LIN {X 0,Y 266.762,Z 400.732,A -85,B 0,C 180,E1 -19209.692,E2 -19209.692} C_VEL
LIN {X 0,Y 260.69,Z 388.855,A -85,B 0,C 180,E1 -19211.354,E2 -19211.354} C_VEL
LIN {X 0,Y 253.783,Z 376.661,A -85,B 0,C 180,E1 -19213.353,E2 -19213.353} C_VEL
LIN {X 0,Y 250.06,Z 370.765,A -85,B 0,C 180,E1 -19214.482,E2 -19214.482} C_VEL
LIN {X 0,Y 247.221,Z 366.216,A -85,B 0,C 180,E1 -19215.384,E2 -19215.384} C_VEL
LIN {X 0,Y 244.284,Z 361.418,A -85,B 0,C 180,E1 -19216.424,E2 -19216.424} C_VEL
LIN {X 0,Y 241.94,Z 353.971,A -85,B 0,C 180,E1 -19220.655,E2 -19220.655} C_VEL
LIN {X 0,Y 241.982,Z 353.963,A -85,B 0,C 180,E1 -19224.489,E2 -19224.489} C_VEL
LIN {X 0,Y 241.941,Z 353.945,A -85,B 0,C 180,E1 -19228.476,E2 -19228.476} C_VEL
LIN {X 0,Y 241.954,Z 353.955,A -85,B 0,C 180,E1 -19232.306,E2 -19232.306} C_VEL
LIN {X 0,Y 242.018,Z 353.954,A -85,B 0,C 180,E1 -19236.012,E2 -19236.012} C_VEL
LIN {X 0,Y 242.013,Z 353.953,A -85,B 0,C 180,E1 -19239.606,E2 -19239.606} C_VEL
LIN {X 0,Y 242.109,Z 353.941,A -85,B 0,C 180,E1 -19243.316,E2 -19243.316} C_VEL
LIN {X 0,Y 242.128,Z 353.949,A -85,B 0,C 180,E1 -19246.573,E2 -19246.573} C_VEL
LIN {X 0,Y 242.36,Z 353.915,A -85,B 0,C 180,E1 -19251.664,E2 -19251.664} C_VEL
LIN {X 0,Y 242.387,Z 353.904,A -85,B 0,C 180,E1 -19253.34,E2 -19253.34} C_VEL
LIN {X 0,Y 242.612,Z 353.876,A -85,B 0,C 180,E1 -19258.341,E2 -19258.341} C_VEL
LIN {X 0,Y 242.612,Z 353.88,A -85,B 0,C 180,E1 -19261.661,E2 -19261.661} C_VEL
LIN {X 0,Y 242.398,Z 353.906,A -85,B 0,C 180,E1 -19266.66,E2 -19266.66} C_VEL
LIN {X 0,Y 242.256,Z 353.934,A -85,B 0,C 180,E1 -19270.025,E2 -19270.025} C_VEL
LIN {X 0,Y 242.116,Z 353.947,A -85,B 0,C 180,E1 -19275.145,E2 -19275.145} C_VEL
LIN {X 0,Y 242.026,Z 353.963,A -85,B 0,C 180,E1 -19278.629,E2 -19278.629} C_VEL
LIN {X 0,Y 241.997,Z 353.965,A -85,B 0,C 180,E1 -19282.182,E2 -19282.182} C_VEL
LIN {X 0,Y 242.063,Z 353.956,A -85,B 0,C 180,E1 -19285.839,E2 -19285.839} C_VEL
LIN {X 0,Y 242.026,Z 353.963,A -85,B 0,C 180,E1 -19289.582,E2 -19289.582} C_VEL
LIN {X 0,Y 241.978,Z 353.965,A -85,B 0,C 180,E1 -19293.494,E2 -19293.494} C_VEL
LIN {X 0,Y 242.004,Z 354.056,A -85,B 0,C 180,E1 -19297.122,E2 -19297.122} C_VEL
LIN {X 0,Y 242.918,Z 356.668,A -85,B 0,C 180,E1 -19297.493,E2 -19297.493} C_VEL
LIN {X 0,Y 245.113,Z 359.008,A -85,B 0,C 180,E1 -19298.192,E2 -19298.192} C_VEL
LIN {X 0,Y 247.682,Z 362.902,A -85,B 0,C 180,E1 -19299.03,E2 -19299.03} C_VEL
LIN {X 0,Y 249.024,Z 364.607,A -85,B 0,C 180,E1 -19299.442,E2 -19299.442} C_VEL
LIN {X 0,Y 255.386,Z 373.693,A -85,B 0,C 180,E1 -19301.336,E2 -19301.336} C_VEL
LIN {X 0,Y 262.149,Z 384.884,A -85,B 0,C 180,E1 -19303.241,E2 -19303.241} C_VEL
LIN {X 0,Y 270.133,Z 399.946,A -85,B 0,C 180,E1 -19305.361,E2 -19305.361} C_VEL
LIN {X 0,Y 275.739,Z 412.188,A -85,B 0,C 180,E1 -19306.793,E2 -19306.793} C_VEL
LIN {X 0,Y 271.981,Z 488.618,A -85,B 0,C 180,E1 -19308.739,E2 -19308.739} C_VEL
LIN {X 0,Y 270.539,Z 503.215,A -85,B 0,C 180,E1 -19309.389,E2 -19309.389} C_VEL
LIN {X 0,Y 268.489,Z 517.743,A -85,B 0,C 180,E1 -19310.355,E2 -19310.355} C_VEL
LIN {X 0,Y 266.247,Z 529.779,A -85,B 0,C 180,E1 -19311.42,E2 -19311.42} C_VEL
LIN {X 0,Y 263.578,Z 541.335,A -85,B 0,C 180,E1 -19312.705,E2 -19312.705} C_VEL
LIN {X 0,Y 260.501,Z 552.94,A -85,B 0,C 180,E1 -19314.328,E2 -19314.328} C_VEL
LIN {X 0,Y 257.523,Z 562.64,A -85,B 0,C 180,E1 -19315.983,E2 -19315.983} C_VEL
LIN {X 0,Y 254.098,Z 573.453,A -85,B 0,C 180,E1 -19318.298,E2 -19318.298} C_VEL
LIN {X 0,Y 251.147,Z 582.347,A -85,B 0,C 180,E1 -19320.679,E2 -19320.679} C_VEL
LIN {X 0,Y 248.431,Z 589.714,A -85,B 0,C 180,E1 -19323.088,E2 -19323.088} C_VEL
LIN {X 0,Y 246.113,Z 595.823,A -85,B 0,C 180,E1 -19325.54,E2 -19325.54} C_VEL
LIN {X 0,Y 244.196,Z 600.861,A -85,B 0,C 180,E1 -19328.029,E2 -19328.029} C_VEL
LIN {X 0,Y 242.228,Z 606.023,A -85,B 0,C 180,E1 -19331.389,E2 -19331.389} C_VEL
LIN {X 0,Y 240.942,Z 609.649,A -85,B 0,C 180,E1 -19334.781,E2 -19334.781} C_VEL
LIN {X 0,Y 240.025,Z 611.858,A -85,B 0,C 180,E1 -19338.173,E2 -19338.173} C_VEL
LIN {X 0,Y 239.773,Z 612.71,A -85,B 0,C 180,E1 -19341.573,E2 -19341.573} C_VEL
LIN {X 0,Y 239.848,Z 612.21,A -85,B 0,C 180,E1 -19345.056,E2 -19345.056} C_VEL
LIN {X 0,Y 239.95,Z 610.455,A -85,B 0,C 180,E1 -19348.322,E2 -19348.322} C_VEL
LIN {X 0,Y 240.27,Z 607.324,A -85,B 0,C 180,E1 -19351.676,E2 -19351.676} C_VEL
LIN {X 0,Y 241.059,Z 602.721,A -85,B 0,C 180,E1 -19355.018,E2 -19355.018} C_VEL
LIN {X 0,Y 242.464,Z 596.49,A -85,B 0,C 180,E1 -19358.333,E2 -19358.333} C_VEL
LIN {X 0,Y 244.301,Z 589.549,A -85,B 0,C 180,E1 -19361.197,E2 -19361.197} C_VEL
LIN {X 0,Y 246.354,Z 581.698,A -85,B 0,C 180,E1 -19363.802,E2 -19363.802} C_VEL
LIN {X 0,Y 248.233,Z 573.619,A -85,B 0,C 180,E1 -19366.024,E2 -19366.024} C_VEL
LIN {X 0,Y 250.756,Z 563.089,A -85,B 0,C 180,E1 -19368.379,E2 -19368.379} C_VEL
LIN {X 0,Y 253.22,Z 552.45,A -85,B 0,C 180,E1 -19370.299,E2 -19370.299} C_VEL
LIN {X 0,Y 255.525,Z 540.847,A -85,B 0,C 180,E1 -19372.008,E2 -19372.008} C_VEL
LIN {X 0,Y 257.784,Z 528.072,A -85,B 0,C 180,E1 -19373.498,E2 -19373.498} C_VEL
LIN {X 0,Y 259.576,Z 515.909,A -85,B 0,C 180,E1 -19374.599,E2 -19374.599} C_VEL
LIN {X 0,Y 261.232,Z 501.809,A -85,B 0,C 180,E1 -19375.549,E2 -19375.549} C_VEL
LIN {X 0,Y 262.272,Z 488.028,A -85,B 0,C 180,E1 -19376.186,E2 -19376.186} C_VEL
LIN {X 0,Y 265.58,Z 403.027,A -85,B 0,C 180,E1 -19378.445,E2 -19378.445} C_VEL
LIN {X 0,Y 263.893,Z 398.103,A -85,B 0,C 180,E1 -19378.83,E2 -19378.83} C_VEL
LIN {X 0,Y 257.563,Z 382.943,A -85,B 0,C 180,E1 -19380.226,E2 -19380.226} C_VEL
LIN {X 0,Y 251.704,Z 370.899,A -85,B 0,C 180,E1 -19381.533,E2 -19381.533} C_VEL
LIN {X 0,Y 243.648,Z 357.672,A -85,B 0,C 180,E1 -19383.35,E2 -19383.35} C_VEL
LIN {X 0,Y 242.306,Z 355.295,A -85,B 0,C 180,E1 -19383.675,E2 -19383.675} C_VEL
LIN {X 0,Y 242.016,Z 353.964,A -85,B 0,C 180,E1 -19383.796,E2 -19383.796} C_VEL
LIN {X 0,Y 242.003,Z 353.966,A -85,B 0,C 180,E1 -19387.578,E2 -19387.578} C_VEL
LIN {X 0,Y 241.938,Z 353.961,A -85,B 0,C 180,E1 -19391.921,E2 -19391.921} C_VEL
LIN {X 0,Y 241.926,Z 353.975,A -85,B 0,C 180,E1 -19396.572,E2 -19396.572} C_VEL
LIN {X 0,Y 241.954,Z 353.971,A -85,B 0,C 180,E1 -19400.279,E2 -19400.279} C_VEL
LIN {X 0,Y 241.984,Z 353.967,A -85,B 0,C 180,E1 -19404.488,E2 -19404.488} C_VEL
LIN {X 0,Y 241.969,Z 353.967,A -85,B 0,C 180,E1 -19408.478,E2 -19408.478} C_VEL
LIN {X 0,Y 241.986,Z 353.946,A -85,B 0,C 180,E1 -19412.309,E2 -19412.309} C_VEL
LIN {X 0,Y 242.032,Z 353.961,A -85,B 0,C 180,E1 -19416.013,E2 -19416.013} C_VEL
LIN {X 0,Y 241.987,Z 353.941,A -85,B 0,C 180,E1 -19419.603,E2 -19419.603} C_VEL
LIN {X 0,Y 242.108,Z 353.952,A -85,B 0,C 180,E1 -19423.317,E2 -19423.317} C_VEL
LIN {X 0,Y 242.157,Z 353.922,A -85,B 0,C 180,E1 -19428.278,E2 -19428.278} C_VEL
LIN {X 0,Y 242.379,Z 353.917,A -85,B 0,C 180,E1 -19431.663,E2 -19431.663} C_VEL
LIN {X 0,Y 242.4,Z 353.906,A -85,B 0,C 180,E1 -19433.34,E2 -19433.34} C_VEL
LIN {X 0,Y 242.61,Z 353.884,A -85,B 0,C 180,E1 -19438.339,E2 -19438.339} C_VEL
LIN {X 0,Y 242.6,Z 353.887,A -85,B 0,C 180,E1 -19439.548,E2 -19439.548} C_VEL
LIN {X 0,Y 241.968,Z 353.976,A -85,B 0,C 180,E1 -19440.929,E2 -19440.929} C_VEL
LIN {X 0,Y 239.092,Z 354.347,A -85,B 0,C 180,E1 -19443.179,E2 -19443.179} C_VEL
LIN {X 0,Y 236.583,Z 354.657,A -85,B 0,C 180,E1 -19445.011,E2 -19445.011} C_VEL
LIN {X 0,Y 235.452,Z 354.786,A -85,B 0,C 180,E1 -19446.436,E2 -19446.436} C_VEL
LIN {X 0,Y 235.332,Z 354.794,A -85,B 0,C 180,E1 -19446.919,E2 -19446.919} C_VEL
LIN {X 0,Y 235.178,Z 354.8,A -85,B 0,C 180,E1 -19450.329,E2 -19450.329} C_VEL
LIN {X 0,Y 235.073,Z 354.812,A -85,B 0,C 180,E1 -19455.609,E2 -19455.609} C_VEL
LIN {X 0,Y 234.982,Z 354.837,A -85,B 0,C 180,E1 -19459.207,E2 -19459.207} C_VEL
LIN {X 0,Y 234.939,Z 354.841,A -85,B 0,C 180,E1 -19462.885,E2 -19462.885} C_VEL
LIN {X 0,Y 234.939,Z 354.834,A -85,B 0,C 180,E1 -19466.661,E2 -19466.661} C_VEL
LIN {X 0,Y 234.892,Z 354.841,A -85,B 0,C 180,E1 -19470.573,E2 -19470.573} C_VEL
LIN {X 0,Y 234.927,Z 354.841,A -85,B 0,C 180,E1 -19474.638,E2 -19474.638} C_VEL
LIN {X 0,Y 234.937,Z 354.846,A -85,B 0,C 180,E1 -19478.945,E2 -19478.945} C_VEL
LIN {X 0,Y 234.882,Z 354.85,A -85,B 0,C 180,E1 -19483.487,E2 -19483.487} C_VEL
LIN {X 0,Y 234.908,Z 355.04,A -85,B 0,C 180,E1 -19486.011,E2 -19486.011} C_VEL
LIN {X 0,Y 236.964,Z 362.224,A -85,B 0,C 180,E1 -19489.237,E2 -19489.237} C_VEL
LIN {X 0,Y 239.314,Z 366.648,A -85,B 0,C 180,E1 -19489.838,E2 -19489.838} C_VEL
LIN {X 0,Y 246.546,Z 381.074,A -85,B 0,C 180,E1 -19491.616,E2 -19491.616} C_VEL
LIN {X 0,Y 254.062,Z 398.232,A -85,B 0,C 180,E1 -19493.393,E2 -19493.393} C_VEL
LIN {X 0,Y 257.193,Z 406.594,A -85,B 0,C 180,E1 -19494.133,E2 -19494.133} C_VEL
LIN {X 0,Y 259.019,Z 420.75,A -85,B 0,C 180,E1 -19494.852,E2 -19494.852} C_VEL
LIN {X 0,Y 255.72,Z 500.655,A -85,B 0,C 180,E1 -19497.01,E2 -19497.01} C_VEL
LIN {X 0,Y 254.462,Z 514.625,A -85,B 0,C 180,E1 -19497.649,E2 -19497.649} C_VEL
LIN {X 0,Y 252.697,Z 528.294,A -85,B 0,C 180,E1 -19498.57,E2 -19498.57} C_VEL
LIN {X 0,Y 250.665,Z 540.694,A -85,B 0,C 180,E1 -19499.691,E2 -19499.691} C_VEL
LIN {X 0,Y 248.233,Z 553.693,A -85,B 0,C 180,E1 -19501.23,E2 -19501.23} C_VEL
LIN {X 0,Y 245.608,Z 565.477,A -85,B 0,C 180,E1 -19502.984,E2 -19502.984} C_VEL
LIN {X 0,Y 243.231,Z 575.273,A -85,B 0,C 180,E1 -19504.775,E2 -19504.775} C_VEL
LIN {X 0,Y 240.52,Z 586.117,A -85,B 0,C 180,E1 -19507.223,E2 -19507.223} C_VEL
LIN {X 0,Y 238.24,Z 595.063,A -85,B 0,C 180,E1 -19509.72,E2 -19509.72} C_VEL
LIN {X 0,Y 236.194,Z 603.633,A -85,B 0,C 180,E1 -19512.69,E2 -19512.69} C_VEL
LIN {X 0,Y 234.835,Z 609.612,A -85,B 0,C 180,E1 -19515.263,E2 -19515.263} C_VEL
LIN {X 0,Y 233.512,Z 615.983,A -85,B 0,C 180,E1 -19518.719,E2 -19518.719} C_VEL
LIN {X 0,Y 233.055,Z 619.631,A -85,B 0,C 180,E1 -19521.328,E2 -19521.328} C_VEL
LIN {X 0,Y 232.742,Z 623.191,A -85,B 0,C 180,E1 -19524.803,E2 -19524.803} C_VEL
LIN {X 0,Y 232.753,Z 625.335,A -85,B 0,C 180,E1 -19528.27,E2 -19528.27} C_VEL
LIN {X 0,Y 232.822,Z 625.893,A -85,B 0,C 180,E1 -19530,E2 -19530} C_VEL
LIN {X 0,Y 232.663,Z 625.992,A -85,B 0,C 180,E1 -19533.463,E2 -19533.463} C_VEL
LIN {X 0,Y 232.813,Z 624.763,A -85,B 0,C 180,E1 -19536.935,E2 -19536.935} C_VEL
LIN {X 0,Y 233.45,Z 622.191,A -85,B 0,C 180,E1 -19540.406,E2 -19540.406} C_VEL
LIN {X 0,Y 234.643,Z 618.189,A -85,B 0,C 180,E1 -19543.863,E2 -19543.863} C_VEL
LIN {X 0,Y 236.101,Z 614.187,A -85,B 0,C 180,E1 -19546.426,E2 -19546.426} C_VEL
LIN {X 0,Y 238.454,Z 607.618,A -85,B 0,C 180,E1 -19549.722,E2 -19549.722} C_VEL
LIN {X 0,Y 241.425,Z 599.911,A -85,B 0,C 180,E1 -19552.687,E2 -19552.687} C_VEL
LIN {X 0,Y 244.327,Z 592.105,A -85,B 0,C 180,E1 -19555.104,E2 -19555.104} C_VEL
LIN {X 0,Y 247.771,Z 582.709,A -85,B 0,C 180,E1 -19557.446,E2 -19557.446} C_VEL
LIN {X 0,Y 251.562,Z 571.263,A -85,B 0,C 180,E1 -19559.727,E2 -19559.727} C_VEL
LIN {X 0,Y 254.627,Z 560.844,A -85,B 0,C 180,E1 -19561.407,E2 -19561.407} C_VEL
LIN {X 0,Y 257.904,Z 548.266,A -85,B 0,C 180,E1 -19563.024,E2 -19563.024} C_VEL
LIN {X 0,Y 260.706,Z 535.983,A -85,B 0,C 180,E1 -19564.244,E2 -19564.244} C_VEL
LIN {X 0,Y 263.268,Z 522.4,A -85,B 0,C 180,E1 -19565.259,E2 -19565.259} C_VEL
LIN {X 0,Y 265.176,Z 508.352,A -85,B 0,C 180,E1 -19566.017,E2 -19566.017} C_VEL
LIN {X 0,Y 266.376,Z 493.63,A -85,B 0,C 180,E1 -19566.532,E2 -19566.532} C_VEL
LIN {X 0,Y 269.746,Z 424.551,A -85,B 0,C 180,E1 -19568.295,E2 -19568.295} C_VEL
LIN {X 0,Y 269.075,Z 420.472,A -85,B 0,C 180,E1 -19568.56,E2 -19568.56} C_VEL
LIN {X 0,Y 261.643,Z 403.746,A -85,B 0,C 180,E1 -19570.603,E2 -19570.603} C_VEL
LIN {X 0,Y 255.013,Z 390.781,A -85,B 0,C 180,E1 -19572.515,E2 -19572.515} C_VEL
LIN {X 0,Y 249.09,Z 380.459,A -85,B 0,C 180,E1 -19574.319,E2 -19574.319} C_VEL
LIN {X 0,Y 243.328,Z 371.168,A -85,B 0,C 180,E1 -19576.191,E2 -19576.191} C_VEL
LIN {X 0,Y 240.05,Z 366.173,A -85,B 0,C 180,E1 -19577.316,E2 -19577.316} C_VEL
LIN {X 0,Y 237.047,Z 361.473,A -85,B 0,C 180,E1 -19578.405,E2 -19578.405} C_VEL
LIN {X 0,Y 234.943,Z 354.839,A -85,B 0,C 180,E1 -19582.313,E2 -19582.313} C_VEL
LIN {X 0,Y 234.934,Z 354.846,A -85,B 0,C 180,E1 -19586.886,E2 -19586.886} C_VEL
LIN {X 0,Y 234.889,Z 354.819,A -85,B 0,C 180,E1 -19591.398,E2 -19591.398} C_VEL
LIN {X 0,Y 234.946,Z 354.833,A -85,B 0,C 180,E1 -19595.243,E2 -19595.243} C_VEL
LIN {X 0,Y 234.963,Z 354.832,A -85,B 0,C 180,E1 -19598.966,E2 -19598.966} C_VEL
LIN {X 0,Y 235.05,Z 354.822,A -85,B 0,C 180,E1 -19603.092,E2 -19603.092} C_VEL
LIN {X 0,Y 235.087,Z 354.813,A -85,B 0,C 180,E1 -19607.921,E2 -19607.921} C_VEL
LIN {X 0,Y 235.297,Z 354.797,A -85,B 0,C 180,E1 -19611.412,E2 -19611.412} C_VEL
LIN {X 0,Y 235.339,Z 354.781,A -85,B 0,C 180,E1 -19613.14,E2 -19613.14} C_VEL
LIN {X 0,Y 235.57,Z 354.753,A -85,B 0,C 180,E1 -19618.291,E2 -19618.291} C_VEL
LIN {X 0,Y 235.571,Z 354.756,A -85,B 0,C 180,E1 -19621.71,E2 -19621.71} C_VEL
LIN {X 0,Y 235.35,Z 354.782,A -85,B 0,C 180,E1 -19626.861,E2 -19626.861} C_VEL
LIN {X 0,Y 235.204,Z 354.812,A -85,B 0,C 180,E1 -19630.329,E2 -19630.329} C_VEL
LIN {X 0,Y 235.065,Z 354.821,A -85,B 0,C 180,E1 -19635.61,E2 -19635.61} C_VEL
LIN {X 0,Y 234.968,Z 354.84,A -85,B 0,C 180,E1 -19639.21,E2 -19639.21} C_VEL
LIN {X 0,Y 234.945,Z 354.845,A -85,B 0,C 180,E1 -19642.885,E2 -19642.885} C_VEL
LIN {X 0,Y 234.965,Z 354.842,A -85,B 0,C 180,E1 -19646.659,E2 -19646.659} C_VEL
LIN {X 0,Y 234.928,Z 354.841,A -85,B 0,C 180,E1 -19650.569,E2 -19650.569} C_VEL
LIN {X 0,Y 234.928,Z 354.838,A -85,B 0,C 180,E1 -19654.639,E2 -19654.639} C_VEL
LIN {X 0,Y 234.913,Z 354.844,A -85,B 0,C 180,E1 -19655.064,E2 -19655.064} C_VEL
LIN {X 0,Y 235.872,Z 357.576,A -85,B 0,C 180,E1 -19655.492,E2 -19655.492} C_VEL
LIN {X 0,Y 238.108,Z 359.896,A -85,B 0,C 180,E1 -19656.272,E2 -19656.272} C_VEL
LIN {X 0,Y 238.796,Z 360.859,A -85,B 0,C 180,E1 -19656.518,E2 -19656.518} C_VEL
LIN {X 0,Y 241.022,Z 364.081,A -85,B 0,C 180,E1 -19657.299,E2 -19657.299} C_VEL
LIN {X 0,Y 242.271,Z 365.585,A -85,B 0,C 180,E1 -19657.713,E2 -19657.713} C_VEL
LIN {X 0,Y 251.05,Z 377.995,A -85,B 0,C 180,E1 -19660.492,E2 -19660.492} C_VEL
LIN {X 0,Y 257.832,Z 389.365,A -85,B 0,C 180,E1 -19662.49,E2 -19662.49} C_VEL
LIN {X 0,Y 265.661,Z 404.415,A -85,B 0,C 180,E1 -19664.662,E2 -19664.662} C_VEL
LIN {X 0,Y 270.194,Z 414.33,A -85,B 0,C 180,E1 -19665.871,E2 -19665.871} C_VEL
LIN {X 0,Y 266.45,Z 488.565,A -85,B 0,C 180,E1 -19667.794,E2 -19667.794} C_VEL
LIN {X 0,Y 265.047,Z 502.54,A -85,B 0,C 180,E1 -19668.411,E2 -19668.411} C_VEL
LIN {X 0,Y 263.205,Z 515.723,A -85,B 0,C 180,E1 -19669.269,E2 -19669.269} C_VEL
LIN {X 0,Y 260.66,Z 529.136,A -85,B 0,C 180,E1 -19670.434,E2 -19670.434} C_VEL
LIN {X 0,Y 257.606,Z 542.009,A -85,B 0,C 180,E1 -19671.885,E2 -19671.885} C_VEL
LIN {X 0,Y 254.216,Z 554.237,A -85,B 0,C 180,E1 -19673.648,E2 -19673.648} C_VEL
LIN {X 0,Y 251.543,Z 562.375,A -85,B 0,C 180,E1 -19675.058,E2 -19675.058} C_VEL
LIN {X 0,Y 248.589,Z 571.627,A -85,B 0,C 180,E1 -19677.029,E2 -19677.029} C_VEL
LIN {X 0,Y 245.365,Z 580.72,A -85,B 0,C 180,E1 -19679.394,E2 -19679.394} C_VEL
LIN {X 0,Y 242.447,Z 588.527,A -85,B 0,C 180,E1 -19681.898,E2 -19681.898} C_VEL
LIN {X 0,Y 239.542,Z 595.808,A -85,B 0,C 180,E1 -19684.823,E2 -19684.823} C_VEL
LIN {X 0,Y 237.492,Z 600.889,A -85,B 0,C 180,E1 -19687.375,E2 -19687.375} C_VEL
LIN {X 0,Y 235.393,Z 606.098,A -85,B 0,C 180,E1 -19690.828,E2 -19690.828} C_VEL
LIN {X 0,Y 234.001,Z 609.765,A -85,B 0,C 180,E1 -19694.318,E2 -19694.318} C_VEL
LIN {X 0,Y 233.006,Z 612.013,A -85,B 0,C 180,E1 -19697.811,E2 -19697.811} C_VEL
LIN {X 0,Y 232.677,Z 612.904,A -85,B 0,C 180,E1 -19701.314,E2 -19701.314} C_VEL
LIN {X 0,Y 232.742,Z 612.47,A -85,B 0,C 180,E1 -19704.803,E2 -19704.803} C_VEL
LIN {X 0,Y 232.856,Z 610.723,A -85,B 0,C 180,E1 -19708.27,E2 -19708.27} C_VEL
LIN {X 0,Y 233.196,Z 607.633,A -85,B 0,C 180,E1 -19711.727,E2 -19711.727} C_VEL
LIN {X 0,Y 234.012,Z 603.09,A -85,B 0,C 180,E1 -19715.169,E2 -19715.169} C_VEL
LIN {X 0,Y 235.474,Z 596.906,A -85,B 0,C 180,E1 -19718.582,E2 -19718.582} C_VEL
LIN {X 0,Y 237.377,Z 590.015,A -85,B 0,C 180,E1 -19721.528,E2 -19721.528} C_VEL
LIN {X 0,Y 239.645,Z 581.461,A -85,B 0,C 180,E1 -19724.444,E2 -19724.444} C_VEL
LIN {X 0,Y 241.852,Z 572.595,A -85,B 0,C 180,E1 -19726.893,E2 -19726.893} C_VEL
LIN {X 0,Y 244.583,Z 561.815,A -85,B 0,C 180,E1 -19729.295,E2 -19729.295} C_VEL
LIN {X 0,Y 247.135,Z 550.878,A -85,B 0,C 180,E1 -19731.258,E2 -19731.258} C_VEL
LIN {X 0,Y 249.612,Z 538.88,A -85,B 0,C 180,E1 -19732.995,E2 -19732.995} C_VEL
LIN {X 0,Y 251.653,Z 527.352,A -85,B 0,C 180,E1 -19734.325,E2 -19734.325} C_VEL
LIN {X 0,Y 253.515,Z 514.93,A -85,B 0,C 180,E1 -19735.447,E2 -19735.447} C_VEL
LIN {X 0,Y 255.154,Z 501.145,A -85,B 0,C 180,E1 -19736.368,E2 -19736.368} C_VEL
LIN {X 0,Y 256.227,Z 486.692,A -85,B 0,C 180,E1 -19737.018,E2 -19737.018} C_VEL
LIN {X 0,Y 259.432,Z 404.138,A -85,B 0,C 180,E1 -19739.262,E2 -19739.262} C_VEL
LIN {X 0,Y 252.867,Z 387.802,A -85,B 0,C 180,E1 -19740.776,E2 -19740.776} C_VEL
LIN {X 0,Y 246.77,Z 375.166,A -85,B 0,C 180,E1 -19742.191,E2 -19742.191} C_VEL
LIN {X 0,Y 238.878,Z 362.146,A -85,B 0,C 180,E1 -19744.046,E2 -19744.046} C_VEL
LIN {X 0,Y 236.884,Z 358.874,A -85,B 0,C 180,E1 -19744.541,E2 -19744.541} C_VEL
LIN {X 0,Y 235.372,Z 356.471,A -85,B 0,C 180,E1 -19744.922,E2 -19744.922} C_VEL
LIN {X 0,Y 234.973,Z 354.828,A -85,B 0,C 180,E1 -19745.086,E2 -19745.086} C_VEL
LIN {X 0,Y 234.942,Z 354.832,A -85,B 0,C 180,E1 -19748.943,E2 -19748.943} C_VEL
LIN {X 0,Y 234.879,Z 354.853,A -85,B 0,C 180,E1 -19753.486,E2 -19753.486} C_VEL
LIN {X 0,Y 234.879,Z 354.852,A -85,B 0,C 180,E1 -19756.511,E2 -19756.511} C_VEL
LIN {X 0,Y 234.916,Z 354.845,A -85,B 0,C 180,E1 -19761.077,E2 -19761.077} C_VEL
LIN {X 0,Y 234.927,Z 354.843,A -85,B 0,C 180,E1 -19765.361,E2 -19765.361} C_VEL
LIN {X 0,Y 234.917,Z 354.848,A -85,B 0,C 180,E1 -19769.429,E2 -19769.429} C_VEL
LIN {X 0,Y 234.989,Z 354.824,A -85,B 0,C 180,E1 -19773.793,E2 -19773.793} C_VEL
LIN {X 0,Y 234.949,Z 354.83,A -85,B 0,C 180,E1 -19778.014,E2 -19778.014} C_VEL
LIN {X 0,Y 235.049,Z 354.832,A -85,B 0,C 180,E1 -19783.092,E2 -19783.092} C_VEL
LIN {X 0,Y 235.089,Z 354.799,A -85,B 0,C 180,E1 -19787.92,E2 -19787.92} C_VEL
LIN {X 0,Y 235.312,Z 354.797,A -85,B 0,C 180,E1 -19791.411,E2 -19791.411} C_VEL
LIN {X 0,Y 235.351,Z 354.784,A -85,B 0,C 180,E1 -19793.139,E2 -19793.139} C_VEL
LIN {X 0,Y 235.569,Z 354.76,A -85,B 0,C 180,E1 -19798.29,E2 -19798.29} C_VEL
LIN {X 0,Y 235.558,Z 354.757,A -85,B 0,C 180,E1 -19801.709,E2 -19801.709} C_VEL
LIN {X 0,Y 235.332,Z 354.794,A -85,B 0,C 180,E1 -19806.919,E2 -19806.919} C_VEL
LIN {X 0,Y 234.581,Z 354.877,A -85,B 0,C 180,E1 -19808.345,E2 -19808.345} C_VEL
LIN {X 0,Y 231.661,Z 355.243,A -85,B 0,C 180,E1 -19810.669,E2 -19810.669} C_VEL
LIN {X 0,Y 229.201,Z 355.561,A -85,B 0,C 180,E1 -19812.563,E2 -19812.563} C_VEL
LIN {X 0,Y 228.119,Z 355.688,A -85,B 0,C 180,E1 -19814.035,E2 -19814.035} C_VEL
LIN {X 0,Y 228.014,Z 355.695,A -85,B 0,C 180,E1 -19814.535,E2 -19814.535} C_VEL
LIN {X 0,Y 227.947,Z 355.713,A -85,B 0,C 180,E1 -19817.957,E2 -19817.957} C_VEL
LIN {X 0,Y 227.913,Z 355.708,A -85,B 0,C 180,E1 -19822.322,E2 -19822.322} C_VEL
LIN {X 0,Y 227.916,Z 355.708,A -85,B 0,C 180,E1 -19826.592,E2 -19826.592} C_VEL
LIN {X 0,Y 227.867,Z 355.716,A -85,B 0,C 180,E1 -19830.281,E2 -19830.281} C_VEL
LIN {X 0,Y 227.872,Z 355.72,A -85,B 0,C 180,E1 -19833.721,E2 -19833.721} C_VEL
LIN {X 0,Y 227.84,Z 355.726,A -85,B 0,C 180,E1 -19838.091,E2 -19838.091} C_VEL
LIN {X 0,Y 227.806,Z 355.72,A -85,B 0,C 180,E1 -19842.743,E2 -19842.743} C_VEL
LIN {X 0,Y 227.867,Z 355.912,A -85,B 0,C 180,E1 -19844.917,E2 -19844.917} C_VEL
LIN {X 0,Y 229.571,Z 361.945,A -85,B 0,C 180,E1 -19847.776,E2 -19847.776} C_VEL
LIN {X 0,Y 237.249,Z 376.315,A -85,B 0,C 180,E1 -19849.819,E2 -19849.819} C_VEL
LIN {X 0,Y 244.298,Z 391.184,A -85,B 0,C 180,E1 -19851.598,E2 -19851.598} C_VEL
LIN {X 0,Y 251.337,Z 408.532,A -85,B 0,C 180,E1 -19853.325,E2 -19853.325} C_VEL
LIN {X 0,Y 253.018,Z 422.042,A -85,B 0,C 180,E1 -19854.03,E2 -19854.03} C_VEL
LIN {X 0,Y 249.647,Z 499.832,A -85,B 0,C 180,E1 -19856.161,E2 -19856.161} C_VEL
LIN {X 0,Y 248.336,Z 514.055,A -85,B 0,C 180,E1 -19856.81,E2 -19856.81} C_VEL
LIN {X 0,Y 246.451,Z 528.394,A -85,B 0,C 180,E1 -19857.799,E2 -19857.799} C_VEL
LIN {X 0,Y 244.184,Z 541.618,A -85,B 0,C 180,E1 -19859.039,E2 -19859.039} C_VEL
LIN {X 0,Y 241.513,Z 555.121,A -85,B 0,C 180,E1 -19860.71,E2 -19860.71} C_VEL
LIN {X 0,Y 238.97,Z 566.025,A -85,B 0,C 180,E1 -19862.407,E2 -19862.407} C_VEL
LIN {X 0,Y 236.278,Z 576.681,A -85,B 0,C 180,E1 -19864.451,E2 -19864.451} C_VEL
LIN {X 0,Y 233.502,Z 587.259,A -85,B 0,C 180,E1 -19866.967,E2 -19866.967} C_VEL
LIN {X 0,Y 231.164,Z 595.98,A -85,B 0,C 180,E1 -19869.536,E2 -19869.536} C_VEL
LIN {X 0,Y 229.127,Z 604.336,A -85,B 0,C 180,E1 -19872.599,E2 -19872.599} C_VEL
LIN {X 0,Y 227.506,Z 611.034,A -85,B 0,C 180,E1 -19875.693,E2 -19875.693} C_VEL
LIN {X 0,Y 226.282,Z 616.969,A -85,B 0,C 180,E1 -19879.26,E2 -19879.26} C_VEL
LIN {X 0,Y 225.758,Z 621.31,A -85,B 0,C 180,E1 -19882.847,E2 -19882.847} C_VEL
LIN {X 0,Y 225.611,Z 624.183,A -85,B 0,C 180,E1 -19886.428,E2 -19886.428} C_VEL
LIN {X 0,Y 225.734,Z 625.67,A -85,B 0,C 180,E1 -19890,E2 -19890} C_VEL
LIN {X 0,Y 225.656,Z 625.901,A -85,B 0,C 180,E1 -19891.785,E2 -19891.785} C_VEL
LIN {X 0,Y 225.591,Z 625.362,A -85,B 0,C 180,E1 -19895.363,E2 -19895.363} C_VEL
LIN {X 0,Y 226.019,Z 623.497,A -85,B 0,C 180,E1 -19898.944,E2 -19898.944} C_VEL
LIN {X 0,Y 226.935,Z 620.263,A -85,B 0,C 180,E1 -19902.52,E2 -19902.52} C_VEL
LIN {X 0,Y 228.738,Z 615.547,A -85,B 0,C 180,E1 -19906.053,E2 -19906.053} C_VEL
LIN {X 0,Y 231.093,Z 609.218,A -85,B 0,C 180,E1 -19909.543,E2 -19909.543} C_VEL
LIN {X 0,Y 233.905,Z 602.198,A -85,B 0,C 180,E1 -19912.525,E2 -19912.525} C_VEL
LIN {X 0,Y 237.377,Z 593.526,A -85,B 0,C 180,E1 -19915.422,E2 -19915.422} C_VEL
LIN {X 0,Y 240.867,Z 584.477,A -85,B 0,C 180,E1 -19917.829,E2 -19917.829} C_VEL
LIN {X 0,Y 244.775,Z 573.541,A -85,B 0,C 180,E1 -19920.162,E2 -19920.162} C_VEL
LIN {X 0,Y 248.131,Z 562.684,A -85,B 0,C 180,E1 -19922.029,E2 -19922.029} C_VEL
LIN {X 0,Y 251.585,Z 550.22,A -85,B 0,C 180,E1 -19923.724,E2 -19923.724} C_VEL
LIN {X 0,Y 254.905,Z 536.507,A -85,B 0,C 180,E1 -19925.137,E2 -19925.137} C_VEL
LIN {X 0,Y 257.522,Z 523.151,A -85,B 0,C 180,E1 -19926.168,E2 -19926.168} C_VEL
LIN {X 0,Y 259.606,Z 508.578,A -85,B 0,C 180,E1 -19926.976,E2 -19926.976} C_VEL
LIN {X 0,Y 260.85,Z 494.139,A -85,B 0,C 180,E1 -19927.497,E2 -19927.497} C_VEL
LIN {X 0,Y 264.334,Z 425.52,A -85,B 0,C 180,E1 -19929.278,E2 -19929.278} C_VEL
LIN {X 0,Y 263.902,Z 423.358,A -85,B 0,C 180,E1 -19929.439,E2 -19929.439} C_VEL
LIN {X 0,Y 256.481,Z 406.499,A -85,B 0,C 180,E1 -19931.585,E2 -19931.585} C_VEL
LIN {X 0,Y 250.54,Z 394.848,A -85,B 0,C 180,E1 -19933.383,E2 -19933.383} C_VEL
LIN {X 0,Y 244.979,Z 385.055,A -85,B 0,C 180,E1 -19935.157,E2 -19935.157} C_VEL
LIN {X 0,Y 239.611,Z 376.227,A -85,B 0,C 180,E1 -19936.984,E2 -19936.984} C_VEL
LIN {X 0,Y 236.12,Z 370.915,A -85,B 0,C 180,E1 -19938.236,E2 -19938.236} C_VEL
LIN {X 0,Y 232.983,Z 366.126,A -85,B 0,C 180,E1 -19939.426,E2 -19939.426} C_VEL
LIN {X 0,Y 229.834,Z 361.521,A -85,B 0,C 180,E1 -19940.677,E2 -19940.677} C_VEL
LIN {X 0,Y 229.463,Z 360.712,A -85,B 0,C 180,E1 -19940.939,E2 -19940.939} C_VEL
LIN {X 0,Y 227.878,Z 355.722,A -85,B 0,C 180,E1 -19944.264,E2 -19944.264} C_VEL
LIN {X 0,Y 227.848,Z 355.7,A -85,B 0,C 180,E1 -19948.375,E2 -19948.375} C_VEL
LIN {X 0,Y 227.845,Z 355.712,A -85,B 0,C 180,E1 -19952.44,E2 -19952.44} C_VEL
LIN {X 0,Y 227.887,Z 355.715,A -85,B 0,C 180,E1 -19956.365,E2 -19956.365} C_VEL
LIN {X 0,Y 227.911,Z 355.71,A -85,B 0,C 180,E1 -19960.172,E2 -19960.172} C_VEL
LIN {X 0,Y 228.017,Z 355.695,A -85,B 0,C 180,E1 -19963.895,E2 -19963.895} C_VEL
LIN {X 0,Y 228.046,Z 355.692,A -85,B 0,C 180,E1 -19967.542,E2 -19967.542} C_VEL
LIN {X 0,Y 228.238,Z 355.679,A -85,B 0,C 180,E1 -19971.144,E2 -19971.144} C_VEL
LIN {X 0,Y 228.291,Z 355.659,A -85,B 0,C 180,E1 -19972.927,E2 -19972.927} C_VEL
LIN {X 0,Y 228.528,Z 355.629,A -85,B 0,C 180,E1 -19978.238,E2 -19978.238} C_VEL
LIN {X 0,Y 228.53,Z 355.632,A -85,B 0,C 180,E1 -19981.763,E2 -19981.763} C_VEL
LIN {X 0,Y 228.302,Z 355.659,A -85,B 0,C 180,E1 -19987.074,E2 -19987.074} C_VEL
LIN {X 0,Y 228.135,Z 355.688,A -85,B 0,C 180,E1 -19990.652,E2 -19990.652} C_VEL
LIN {X 0,Y 228.026,Z 355.707,A -85,B 0,C 180,E1 -19994.275,E2 -19994.275} C_VEL
LIN {X 0,Y 227.925,Z 355.715,A -85,B 0,C 180,E1 -19997.96,E2 -19997.96} C_VEL
LIN {X 0,Y 227.908,Z 355.721,A -85,B 0,C 180,E1 -20002.319,E2 -20002.319} C_VEL
LIN {X 0,Y 227.939,Z 355.717,A -85,B 0,C 180,E1 -20006.603,E2 -20006.603} C_VEL
LIN {X 0,Y 227.905,Z 355.718,A -85,B 0,C 180,E1 -20010.297,E2 -20010.297} C_VEL
LIN {X 0,Y 227.909,Z 355.719,A -85,B 0,C 180,E1 -20012.792,E2 -20012.792} C_VEL
LIN {X 0,Y 228.798,Z 358.391,A -85,B 0,C 180,E1 -20013.249,E2 -20013.249} C_VEL
LIN {X 0,Y 230.806,Z 360.631,A -85,B 0,C 180,E1 -20014.037,E2 -20014.037} C_VEL
LIN {X 0,Y 231.756,Z 361.484,A -85,B 0,C 180,E1 -20014.39,E2 -20014.39} C_VEL
LIN {X 0,Y 233.91,Z 364.801,A -85,B 0,C 180,E1 -20015.237,E2 -20015.237} C_VEL
LIN {X 0,Y 235.506,Z 366.557,A -85,B 0,C 180,E1 -20015.81,E2 -20015.81} C_VEL
LIN {X 0,Y 238.284,Z 370.314,A -85,B 0,C 180,E1 -20016.806,E2 -20016.806} C_VEL
LIN {X 0,Y 247.132,Z 382.941,A -85,B 0,C 180,E1 -20019.736,E2 -20019.736} C_VEL
LIN {X 0,Y 253.858,Z 394.428,A -85,B 0,C 180,E1 -20021.804,E2 -20021.804} C_VEL
LIN {X 0,Y 261.459,Z 409.345,A -85,B 0,C 180,E1 -20024.003,E2 -20024.003} C_VEL
LIN {X 0,Y 264.779,Z 416.648,A -85,B 0,C 180,E1 -20024.928,E2 -20024.928} C_VEL
LIN {X 0,Y 260.888,Z 489.465,A -85,B 0,C 180,E1 -20026.841,E2 -20026.841} C_VEL
LIN {X 0,Y 259.383,Z 503.663,A -85,B 0,C 180,E1 -20027.494,E2 -20027.494} C_VEL
LIN {X 0,Y 257.386,Z 517.131,A -85,B 0,C 180,E1 -20028.406,E2 -20028.406} C_VEL
LIN {X 0,Y 255.152,Z 528.493,A -85,B 0,C 180,E1 -20029.404,E2 -20029.404} C_VEL
LIN {X 0,Y 251.981,Z 541.53,A -85,B 0,C 180,E1 -20030.875,E2 -20030.875} C_VEL
LIN {X 0,Y 248.717,Z 553.013,A -85,B 0,C 180,E1 -20032.524,E2 -20032.524} C_VEL
LIN {X 0,Y 245.013,Z 564.08,A -85,B 0,C 180,E1 -20034.491,E2 -20034.491} C_VEL
LIN {X 0,Y 241.324,Z 574.72,A -85,B 0,C 180,E1 -20036.905,E2 -20036.905} C_VEL
LIN {X 0,Y 238.023,Z 583.687,A -85,B 0,C 180,E1 -20039.46,E2 -20039.46} C_VEL
LIN {X 0,Y 234.69,Z 591.819,A -85,B 0,C 180,E1 -20042.345,E2 -20042.345} C_VEL
LIN {X 0,Y 231.805,Z 598.627,A -85,B 0,C 180,E1 -20045.446,E2 -20045.446} C_VEL
LIN {X 0,Y 229.593,Z 603.752,A -85,B 0,C 180,E1 -20048.45,E2 -20048.45} C_VEL
LIN {X 0,Y 227.703,Z 608.213,A -85,B 0,C 180,E1 -20052.023,E2 -20052.023} C_VEL
LIN {X 0,Y 226.45,Z 611.197,A -85,B 0,C 180,E1 -20055.624,E2 -20055.624} C_VEL
LIN {X 0,Y 225.725,Z 612.8,A -85,B 0,C 180,E1 -20059.234,E2 -20059.234} C_VEL
LIN {X 0,Y 225.573,Z 613.064,A -85,B 0,C 180,E1 -20062.841,E2 -20062.841} C_VEL
LIN {X 0,Y 225.688,Z 612.543,A -85,B 0,C 180,E1 -20065.209,E2 -20065.209} C_VEL
LIN {X 0,Y 225.763,Z 610.992,A -85,B 0,C 180,E1 -20068.216,E2 -20068.216} C_VEL
LIN {X 0,Y 226.123,Z 607.939,A -85,B 0,C 180,E1 -20071.781,E2 -20071.781} C_VEL
LIN {X 0,Y 226.968,Z 603.452,A -85,B 0,C 180,E1 -20075.33,E2 -20075.33} C_VEL
LIN {X 0,Y 228.491,Z 597.321,A -85,B 0,C 180,E1 -20078.846,E2 -20078.846} C_VEL
LIN {X 0,Y 230.461,Z 590.479,A -85,B 0,C 180,E1 -20081.879,E2 -20081.879} C_VEL
LIN {X 0,Y 232.574,Z 582.951,A -85,B 0,C 180,E1 -20084.568,E2 -20084.568} C_VEL
LIN {X 0,Y 234.678,Z 574.791,A -85,B 0,C 180,E1 -20086.976,E2 -20086.976} C_VEL
LIN {X 0,Y 237.417,Z 564.41,A -85,B 0,C 180,E1 -20089.452,E2 -20089.452} C_VEL
LIN {X 0,Y 240.292,Z 552.795,A -85,B 0,C 180,E1 -20091.669,E2 -20091.669} C_VEL
LIN {X 0,Y 242.805,Z 541.175,A -85,B 0,C 180,E1 -20093.452,E2 -20093.452} C_VEL
LIN {X 0,Y 245.228,Z 528.383,A -85,B 0,C 180,E1 -20095.006,E2 -20095.006} C_VEL
LIN {X 0,Y 247.185,Z 516.186,A -85,B 0,C 180,E1 -20096.148,E2 -20096.148} C_VEL
LIN {X 0,Y 248.956,Z 502.043,A -85,B 0,C 180,E1 -20097.134,E2 -20097.134} C_VEL
LIN {X 0,Y 250.049,Z 488.168,A -85,B 0,C 180,E1 -20097.799,E2 -20097.799} C_VEL
LIN {X 0,Y 253.444,Z 406.097,A -85,B 0,C 180,E1 -20100.074,E2 -20100.074} C_VEL
LIN {X 0,Y 247.497,Z 391.21,A -85,B 0,C 180,E1 -20101.51,E2 -20101.51} C_VEL
LIN {X 0,Y 241.691,Z 379.073,A -85,B 0,C 180,E1 -20102.919,E2 -20102.919} C_VEL
LIN {X 0,Y 234.033,Z 366.357,A -85,B 0,C 180,E1 -20104.802,E2 -20104.802} C_VEL
LIN {X 0,Y 229.984,Z 359.873,A -85,B 0,C 180,E1 -20105.859,E2 -20105.859} C_VEL
LIN {X 0,Y 228.294,Z 357.303,A -85,B 0,C 180,E1 -20106.311,E2 -20106.311} C_VEL
LIN {X 0,Y 227.913,Z 355.709,A -85,B 0,C 180,E1 -20106.488,E2 -20106.488} C_VEL
LIN {X 0,Y 227.832,Z 355.707,A -85,B 0,C 180,E1 -20110.374,E2 -20110.374} C_VEL
LIN {X 0,Y 227.827,Z 355.725,A -85,B 0,C 180,E1 -20115.193,E2 -20115.193} C_VEL
LIN {X 0,Y 227.823,Z 355.73,A -85,B 0,C 180,E1 -20119.622,E2 -20119.622} C_VEL
LIN {X 0,Y 227.878,Z 355.724,A -85,B 0,C 180,E1 -20124.127,E2 -20124.127} C_VEL
LIN {X 0,Y 227.863,Z 355.724,A -85,B 0,C 180,E1 -20128.376,E2 -20128.376} C_VEL
LIN {X 0,Y 227.87,Z 355.703,A -85,B 0,C 180,E1 -20132.442,E2 -20132.442} C_VEL
LIN {X 0,Y 227.896,Z 355.722,A -85,B 0,C 180,E1 -20136.365,E2 -20136.365} C_VEL
LIN {X 0,Y 227.892,Z 355.697,A -85,B 0,C 180,E1 -20140.169,E2 -20140.169} C_VEL
LIN {X 0,Y 228.012,Z 355.706,A -85,B 0,C 180,E1 -20143.894,E2 -20143.894} C_VEL
LIN {X 0,Y 228.134,Z 355.678,A -85,B 0,C 180,E1 -20149.348,E2 -20149.348} C_VEL
LIN {X 0,Y 228.303,Z 355.663,A -85,B 0,C 180,E1 -20152.926,E2 -20152.926} C_VEL
LIN {X 0,Y 228.528,Z 355.637,A -85,B 0,C 180,E1 -20158.237,E2 -20158.237} C_VEL
LIN {X 0,Y 228.491,Z 355.636,A -85,B 0,C 180,E1 -20161.762,E2 -20161.762} C_VEL
LIN {X 0,Y 228.289,Z 355.671,A -85,B 0,C 180,E1 -20167.073,E2 -20167.073} C_VEL
LIN {X 0,Y 228.12,Z 355.681,A -85,B 0,C 180,E1 -20170.652,E2 -20170.652} C_VEL
LIN {X 0,Y 228.014,Z 355.695,A -85,B 0,C 180,E1 -20174.535,E2 -20174.535} C_VEL
LIN {X 0,Y 227.277,Z 355.786,A -85,B 0,C 180,E1 -20176.007,E2 -20176.007} C_VEL
LIN {X 0,Y 224.336,Z 356.166,A -85,B 0,C 180,E1 -20178.408,E2 -20178.408} C_VEL
LIN {X 0,Y 221.902,Z 356.458,A -85,B 0,C 180,E1 -20180.368,E2 -20180.368} C_VEL
LIN {X 0,Y 220.911,Z 356.577,A -85,B 0,C 180,E1 -20181.891,E2 -20181.891} C_VEL
LIN {X 0,Y 220.857,Z 356.587,A -85,B 0,C 180,E1 -20182.407,E2 -20182.407} C_VEL
LIN {X 0,Y 220.859,Z 356.589,A -85,B 0,C 180,E1 -20187.005,E2 -20187.005} C_VEL
LIN {X 0,Y 220.813,Z 356.595,A -85,B 0,C 180,E1 -20190.759,E2 -20190.759} C_VEL
LIN {X 0,Y 220.797,Z 356.602,A -85,B 0,C 180,E1 -20194.955,E2 -20194.955} C_VEL
LIN {X 0,Y 220.802,Z 356.602,A -85,B 0,C 180,E1 -20199.537,E2 -20199.537} C_VEL
LIN {X 0,Y 220.758,Z 356.77,A -85,B 0,C 180,E1 -20203.718,E2 -20203.718} C_VEL
LIN {X 0,Y 222.297,Z 361.87,A -85,B 0,C 180,E1 -20206.219,E2 -20206.219} C_VEL
LIN {X 0,Y 230.114,Z 376.004,A -85,B 0,C 180,E1 -20208.44,E2 -20208.44} C_VEL
LIN {X 0,Y 235.949,Z 387.796,A -85,B 0,C 180,E1 -20210.009,E2 -20210.009} C_VEL
LIN {X 0,Y 242.773,Z 403.62,A -85,B 0,C 180,E1 -20211.784,E2 -20211.784} C_VEL
LIN {X 0,Y 245.882,Z 412.159,A -85,B 0,C 180,E1 -20212.594,E2 -20212.594} C_VEL
LIN {X 0,Y 247.065,Z 423.105,A -85,B 0,C 180,E1 -20213.16,E2 -20213.16} C_VEL
LIN {X 0,Y 243.57,Z 500.321,A -85,B 0,C 180,E1 -20215.323,E2 -20215.323} C_VEL
LIN {X 0,Y 242.12,Z 515.031,A -85,B 0,C 180,E1 -20216.03,E2 -20216.03} C_VEL
LIN {X 0,Y 240.261,Z 528.495,A -85,B 0,C 180,E1 -20216.99,E2 -20216.99} C_VEL
LIN {X 0,Y 237.732,Z 542.541,A -85,B 0,C 180,E1 -20218.35,E2 -20218.35} C_VEL
LIN {X 0,Y 235.349,Z 554.224,A -85,B 0,C 180,E1 -20219.836,E2 -20219.836} C_VEL
LIN {X 0,Y 232.69,Z 565.391,A -85,B 0,C 180,E1 -20221.596,E2 -20221.596} C_VEL
LIN {X 0,Y 229.832,Z 576.116,A -85,B 0,C 180,E1 -20223.68,E2 -20223.68} C_VEL
LIN {X 0,Y 226.919,Z 586.754,A -85,B 0,C 180,E1 -20226.258,E2 -20226.258} C_VEL
LIN {X 0,Y 224.47,Z 595.526,A -85,B 0,C 180,E1 -20228.897,E2 -20228.897} C_VEL
LIN {X 0,Y 222.227,Z 603.936,A -85,B 0,C 180,E1 -20232.041,E2 -20232.041} C_VEL
LIN {X 0,Y 220.575,Z 610.681,A -85,B 0,C 180,E1 -20235.233,E2 -20235.233} C_VEL
LIN {X 0,Y 219.261,Z 616.652,A -85,B 0,C 180,E1 -20238.912,E2 -20238.912} C_VEL
LIN {X 0,Y 218.946,Z 619.032,A -85,B 0,C 180,E1 -20240.765,E2 -20240.765} C_VEL
LIN {X 0,Y 218.565,Z 622.656,A -85,B 0,C 180,E1 -20244.465,E2 -20244.465} C_VEL
LIN {X 0,Y 218.564,Z 624.859,A -85,B 0,C 180,E1 -20248.157,E2 -20248.157} C_VEL
LIN {X 0,Y 218.648,Z 625.447,A -85,B 0,C 180,E1 -20250,E2 -20250} C_VEL
LIN {X 0,Y 218.497,Z 625.603,A -85,B 0,C 180,E1 -20253.688,E2 -20253.688} C_VEL
LIN {X 0,Y 218.68,Z 624.431,A -85,B 0,C 180,E1 -20257.386,E2 -20257.386} C_VEL
LIN {X 0,Y 219.395,Z 621.922,A -85,B 0,C 180,E1 -20261.081,E2 -20261.081} C_VEL
LIN {X 0,Y 220.845,Z 618.007,A -85,B 0,C 180,E1 -20264.749,E2 -20264.749} C_VEL
LIN {X 0,Y 223.066,Z 612.539,A -85,B 0,C 180,E1 -20268.364,E2 -20268.364} C_VEL
LIN {X 0,Y 225.159,Z 607.368,A -85,B 0,C 180,E1 -20271.035,E2 -20271.035} C_VEL
LIN {X 0,Y 228.324,Z 599.954,A -85,B 0,C 180,E1 -20274.069,E2 -20274.069} C_VEL
LIN {X 0,Y 232.067,Z 590.764,A -85,B 0,C 180,E1 -20277.017,E2 -20277.017} C_VEL
LIN {X 0,Y 235.884,Z 581.181,A -85,B 0,C 180,E1 -20279.445,E2 -20279.445} C_VEL
LIN {X 0,Y 239.701,Z 570.487,A -85,B 0,C 180,E1 -20281.627,E2 -20281.627} C_VEL
LIN {X 0,Y 243.393,Z 558.875,A -85,B 0,C 180,E1 -20283.519,E2 -20283.519} C_VEL
LIN {X 0,Y 246.593,Z 547.447,A -85,B 0,C 180,E1 -20284.998,E2 -20284.998} C_VEL
LIN {X 0,Y 249.612,Z 535.057,A -85,B 0,C 180,E1 -20286.246,E2 -20286.246} C_VEL
LIN {X 0,Y 252.319,Z 521.32,A -85,B 0,C 180,E1 -20287.286,E2 -20287.286} C_VEL
LIN {X 0,Y 254.38,Z 506.996,A -85,B 0,C 180,E1 -20288.056,E2 -20288.056} C_VEL
LIN {X 0,Y 255.548,Z 493.156,A -85,B 0,C 180,E1 -20288.54,E2 -20288.54} C_VEL
LIN {X 0,Y 259.049,Z 427.094,A -85,B 0,C 180,E1 -20290.271,E2 -20290.271} C_VEL
LIN {X 0,Y 253.584,Z 414.057,A -85,B 0,C 180,E1 -20291.927,E2 -20291.927} C_VEL
LIN {X 0,Y 247.972,Z 402.483,A -85,B 0,C 180,E1 -20293.684,E2 -20293.684} C_VEL
LIN {X 0,Y 241.729,Z 390.926,A -85,B 0,C 180,E1 -20295.752,E2 -20295.752} C_VEL
LIN {X 0,Y 235.756,Z 381.043,A -85,B 0,C 180,E1 -20297.867,E2 -20297.867} C_VEL
LIN {X 0,Y 232.31,Z 375.689,A -85,B 0,C 180,E1 -20299.168,E2 -20299.168} C_VEL
LIN {X 0,Y 229.437,Z 371.265,A -85,B 0,C 180,E1 -20300.311,E2 -20300.311} C_VEL
LIN {X 0,Y 225.721,Z 365.864,A -85,B 0,C 180,E1 -20301.865,E2 -20301.865} C_VEL
LIN {X 0,Y 222.233,Z 360.906,A -85,B 0,C 180,E1 -20303.422,E2 -20303.422} C_VEL
LIN {X 0,Y 222.049,Z 360.395,A -85,B 0,C 180,E1 -20303.598,E2 -20303.598} C_VEL
LIN {X 0,Y 220.833,Z 356.6,A -85,B 0,C 180,E1 -20306.375,E2 -20306.375} C_VEL
LIN {X 0,Y 220.829,Z 356.563,A -85,B 0,C 180,E1 -20309.389,E2 -20309.389} C_VEL
LIN {X 0,Y 220.868,Z 356.597,A -85,B 0,C 180,E1 -20313.547,E2 -20313.547} C_VEL
LIN {X 0,Y 220.86,Z 356.6,A -85,B 0,C 180,E1 -20317.552,E2 -20317.552} C_VEL
LIN {X 0,Y 220.923,Z 356.584,A -85,B 0,C 180,E1 -20322.617,E2 -20322.617} C_VEL
LIN {X 0,Y 220.986,Z 356.575,A -85,B 0,C 180,E1 -20327.138,E2 -20327.138} C_VEL
LIN {X 0,Y 221.18,Z 356.56,A -85,B 0,C 180,E1 -20330.859,E2 -20330.859} C_VEL
LIN {X 0,Y 221.228,Z 356.539,A -85,B 0,C 180,E1 -20332.7,E2 -20332.7} C_VEL
LIN {X 0,Y 221.462,Z 356.509,A -85,B 0,C 180,E1 -20338.182,E2 -20338.182} C_VEL
LIN {X 0,Y 221.464,Z 356.512,A -85,B 0,C 180,E1 -20341.819,E2 -20341.819} C_VEL
LIN {X 0,Y 221.239,Z 356.537,A -85,B 0,C 180,E1 -20347.301,E2 -20347.301} C_VEL
LIN {X 0,Y 221.055,Z 356.565,A -85,B 0,C 180,E1 -20350.998,E2 -20350.998} C_VEL
LIN {X 0,Y 220.971,Z 356.572,A -85,B 0,C 180,E1 -20356.634,E2 -20356.634} C_VEL
LIN {X 0,Y 220.856,Z 356.588,A -85,B 0,C 180,E1 -20360.49,E2 -20360.49} C_VEL
LIN {X 0,Y 220.857,Z 356.589,A -85,B 0,C 180,E1 -20364.437,E2 -20364.437} C_VEL
LIN {X 0,Y 220.832,Z 356.594,A -85,B 0,C 180,E1 -20368.515,E2 -20368.515} C_VEL
LIN {X 0,Y 220.874,Z 356.594,A -85,B 0,C 180,E1 -20370.209,E2 -20370.209} C_VEL
LIN {X 0,Y 221.777,Z 359.347,A -85,B 0,C 180,E1 -20370.751,E2 -20370.751} C_VEL
LIN {X 0,Y 223.737,Z 361.491,A -85,B 0,C 180,E1 -20371.614,E2 -20371.614} C_VEL
LIN {X 0,Y 224.899,Z 362.397,A -85,B 0,C 180,E1 -20372.09,E2 -20372.09} C_VEL
LIN {X 0,Y 226.933,Z 365.691,A -85,B 0,C 180,E1 -20372.989,E2 -20372.989} C_VEL
LIN {X 0,Y 228.77,Z 367.503,A -85,B 0,C 180,E1 -20373.711,E2 -20373.711} C_VEL
LIN {X 0,Y 231.39,Z 371.147,A -85,B 0,C 180,E1 -20374.754,E2 -20374.754} C_VEL
LIN {X 0,Y 236.152,Z 377.674,A -85,B 0,C 180,E1 -20376.529,E2 -20376.529} C_VEL
LIN {X 0,Y 243.565,Z 388.378,A -85,B 0,C 180,E1 -20379.057,E2 -20379.057} C_VEL
LIN {X 0,Y 249.923,Z 399.504,A -85,B 0,C 180,E1 -20381.097,E2 -20381.097} C_VEL
LIN {X 0,Y 256.926,Z 413.496,A -85,B 0,C 180,E1 -20383.214,E2 -20383.214} C_VEL
LIN {X 0,Y 259.466,Z 419.14,A -85,B 0,C 180,E1 -20383.957,E2 -20383.957} C_VEL
LIN {X 0,Y 255.495,Z 489.536,A -85,B 0,C 180,E1 -20385.817,E2 -20385.817} C_VEL
LIN {X 0,Y 253.924,Z 503.971,A -85,B 0,C 180,E1 -20386.492,E2 -20386.492} C_VEL
LIN {X 0,Y 251.846,Z 517.408,A -85,B 0,C 180,E1 -20387.414,E2 -20387.414} C_VEL
LIN {X 0,Y 249.319,Z 529.644,A -85,B 0,C 180,E1 -20388.515,E2 -20388.515} C_VEL
LIN {X 0,Y 246.033,Z 542.495,A -85,B 0,C 180,E1 -20390.007,E2 -20390.007} C_VEL
LIN {X 0,Y 242.468,Z 554.501,A -85,B 0,C 180,E1 -20391.796,E2 -20391.796} C_VEL
LIN {X 0,Y 239.155,Z 563.816,A -85,B 0,C 180,E1 -20393.483,E2 -20393.483} C_VEL
LIN {X 0,Y 235.333,Z 574.535,A -85,B 0,C 180,E1 -20395.949,E2 -20395.949} C_VEL
LIN {X 0,Y 231.905,Z 583.227,A -85,B 0,C 180,E1 -20398.438,E2 -20398.438} C_VEL
LIN {X 0,Y 228.799,Z 590.645,A -85,B 0,C 180,E1 -20401.068,E2 -20401.068} C_VEL
LIN {X 0,Y 225.714,Z 597.599,A -85,B 0,C 180,E1 -20404.157,E2 -20404.157} C_VEL
LIN {X 0,Y 223.517,Z 602.387,A -85,B 0,C 180,E1 -20406.857,E2 -20406.857} C_VEL
LIN {X 0,Y 221.294,Z 607.315,A -85,B 0,C 180,E1 -20410.521,E2 -20410.521} C_VEL
LIN {X 0,Y 220.126,Z 610,A -85,B 0,C 180,E1 -20413.301,E2 -20413.301} C_VEL
LIN {X 0,Y 219.008,Z 612.324,A -85,B 0,C 180,E1 -20417.019,E2 -20417.019} C_VEL
LIN {X 0,Y 218.514,Z 613.292,A -85,B 0,C 180,E1 -20420.746,E2 -20420.746} C_VEL
LIN {X 0,Y 218.553,Z 612.931,A -85,B 0,C 180,E1 -20424.464,E2 -20424.464} C_VEL
LIN {X 0,Y 218.673,Z 611.259,A -85,B 0,C 180,E1 -20428.158,E2 -20428.158} C_VEL
LIN {X 0,Y 219.054,Z 608.245,A -85,B 0,C 180,E1 -20431.838,E2 -20431.838} C_VEL
LIN {X 0,Y 219.929,Z 603.803,A -85,B 0,C 180,E1 -20435.501,E2 -20435.501} C_VEL
LIN {X 0,Y 221.089,Z 599.389,A -85,B 0,C 180,E1 -20438.224,E2 -20438.224} C_VEL
LIN {X 0,Y 222.952,Z 593.021,A -85,B 0,C 180,E1 -20441.362,E2 -20441.362} C_VEL
LIN {X 0,Y 225.257,Z 585.124,A -85,B 0,C 180,E1 -20444.453,E2 -20444.453} C_VEL
LIN {X 0,Y 227.496,Z 576.878,A -85,B 0,C 180,E1 -20447.066,E2 -20447.066} C_VEL
LIN {X 0,Y 230.274,Z 566.941,A -85,B 0,C 180,E1 -20449.616,E2 -20449.616} C_VEL
LIN {X 0,Y 233.174,Z 555.871,A -85,B 0,C 180,E1 -20451.899,E2 -20451.899} C_VEL
LIN {X 0,Y 236.062,Z 543.457,A -85,B 0,C 180,E1 -20453.931,E2 -20453.931} C_VEL
LIN {X 0,Y 238.533,Z 531.162,A -85,B 0,C 180,E1 -20455.524,E2 -20455.524} C_VEL
LIN {X 0,Y 240.882,Z 517.445,A -85,B 0,C 180,E1 -20456.886,E2 -20456.886} C_VEL
LIN {X 0,Y 242.705,Z 503.673,A -85,B 0,C 180,E1 -20457.893,E2 -20457.893} C_VEL
LIN {X 0,Y 243.935,Z 489.399,A -85,B 0,C 180,E1 -20458.618,E2 -20458.618} C_VEL
LIN {X 0,Y 247.34,Z 413.611,A -85,B 0,C 180,E1 -20460.76,E2 -20460.76} C_VEL
LIN {X 0,Y 247.487,Z 407.928,A -85,B 0,C 180,E1 -20460.933,E2 -20460.933} C_VEL
LIN {X 0,Y 241.661,Z 393.448,A -85,B 0,C 180,E1 -20462.406,E2 -20462.406} C_VEL
LIN {X 0,Y 236.408,Z 382.464,A -85,B 0,C 180,E1 -20463.743,E2 -20463.743} C_VEL
LIN {X 0,Y 227.508,Z 367.838,A -85,B 0,C 180,E1 -20466.051,E2 -20466.051} C_VEL
LIN {X 0,Y 225.155,Z 364.222,A -85,B 0,C 180,E1 -20466.695,E2 -20466.695} C_VEL
LIN {X 0,Y 223.211,Z 361.069,A -85,B 0,C 180,E1 -20467.249,E2 -20467.249} C_VEL
LIN {X 0,Y 221.358,Z 358.557,A -85,B 0,C 180,E1 -20467.769,E2 -20467.769} C_VEL
LIN {X 0,Y 220.832,Z 356.603,A -85,B 0,C 180,E1 -20467.982,E2 -20467.982} C_VEL
LIN {X 0,Y 220.771,Z 356.596,A -85,B 0,C 180,E1 -20471.951,E2 -20471.951} C_VEL
LIN {X 0,Y 220.768,Z 356.605,A -85,B 0,C 180,E1 -20475.543,E2 -20475.543} C_VEL
LIN {X 0,Y 220.804,Z 356.606,A -85,B 0,C 180,E1 -20480.462,E2 -20480.462} C_VEL
LIN {X 0,Y 220.799,Z 356.605,A -85,B 0,C 180,E1 -20485.044,E2 -20485.044} C_VEL
LIN {X 0,Y 220.831,Z 356.603,A -85,B 0,C 180,E1 -20489.388,E2 -20489.388} C_VEL
LIN {X 0,Y 220.888,Z 356.576,A -85,B 0,C 180,E1 -20493.548,E2 -20493.548} C_VEL
LIN {X 0,Y 220.849,Z 356.592,A -85,B 0,C 180,E1 -20497.55,E2 -20497.55} C_VEL
LIN {X 0,Y 220.916,Z 356.588,A -85,B 0,C 180,E1 -20502.624,E2 -20502.624} C_VEL
LIN {X 0,Y 220.979,Z 356.554,A -85,B 0,C 180,E1 -20507.136,E2 -20507.136} C_VEL
LIN {X 0,Y 221.191,Z 356.557,A -85,B 0,C 180,E1 -20510.858,E2 -20510.858} C_VEL
LIN {X 0,Y 221.24,Z 356.545,A -85,B 0,C 180,E1 -20512.699,E2 -20512.699} C_VEL
LIN {X 0,Y 221.462,Z 356.517,A -85,B 0,C 180,E1 -20518.181,E2 -20518.181} C_VEL
LIN {X 0,Y 221.428,Z 356.514,A -85,B 0,C 180,E1 -20521.818,E2 -20521.818} C_VEL
LIN {X 0,Y 221.227,Z 356.551,A -85,B 0,C 180,E1 -20527.3,E2 -20527.3} C_VEL
LIN {X 0,Y 221.046,Z 356.566,A -85,B 0,C 180,E1 -20530.997,E2 -20530.997} C_VEL
LIN {X 0,Y 220.96,Z 356.573,A -85,B 0,C 180,E1 -20534.741,E2 -20534.741} C_VEL
LIN {X 0,Y 220.882,Z 356.595,A -85,B 0,C 180,E1 -20538.552,E2 -20538.552} C_VEL
LIN {X 0,Y 220.857,Z 356.587,A -85,B 0,C 180,E1 -20542.407,E2 -20542.407} C_VEL
LIN {X 0,Y 220.242,Z 356.675,A -85,B 0,C 180,E1 -20543.929,E2 -20543.929} C_VEL
LIN {X 0,Y 218.653,Z 356.875,A -85,B 0,C 180,E1 -20545.424,E2 -20545.424} C_VEL
LIN {X 0,Y 214.859,Z 357.345,A -85,B 0,C 180,E1 -20548.439,E2 -20548.439} C_VEL
LIN {X 0,Y 213.807,Z 357.468,A -85,B 0,C 180,E1 -20550.016,E2 -20550.016} C_VEL
LIN {X 0,Y 213.732,Z 357.476,A -85,B 0,C 180,E1 -20550.551,E2 -20550.551} C_VEL
LIN {X 0,Y 213.767,Z 357.477,A -85,B 0,C 180,E1 -20554.725,E2 -20554.725} C_VEL
LIN {X 0,Y 213.719,Z 357.489,A -85,B 0,C 180,E1 -20558.667,E2 -20558.667} C_VEL
LIN {X 0,Y 213.721,Z 357.54,A -85,B 0,C 180,E1 -20562.385,E2 -20562.385} C_VEL
LIN {X 0,Y 214.818,Z 361.48,A -85,B 0,C 180,E1 -20564.451,E2 -20564.451} C_VEL
LIN {X 0,Y 217.519,Z 366.018,A -85,B 0,C 180,E1 -20565.301,E2 -20565.301} C_VEL
LIN {X 0,Y 223.907,Z 377.524,A -85,B 0,C 180,E1 -20567.219,E2 -20567.219} C_VEL
LIN {X 0,Y 230.629,Z 390.909,A -85,B 0,C 180,E1 -20569.122,E2 -20569.122} C_VEL
LIN {X 0,Y 237.549,Z 407.167,A -85,B 0,C 180,E1 -20571.015,E2 -20571.015} C_VEL
LIN {X 0,Y 240.111,Z 413.87,A -85,B 0,C 180,E1 -20571.701,E2 -20571.701} C_VEL
LIN {X 0,Y 241.181,Z 423.872,A -85,B 0,C 180,E1 -20572.239,E2 -20572.239} C_VEL
LIN {X 0,Y 237.541,Z 500.727,A -85,B 0,C 180,E1 -20574.441,E2 -20574.441} C_VEL
LIN {X 0,Y 236.038,Z 515.234,A -85,B 0,C 180,E1 -20575.16,E2 -20575.16} C_VEL
LIN {X 0,Y 233.943,Z 529.736,A -85,B 0,C 180,E1 -20576.238,E2 -20576.238} C_VEL
LIN {X 0,Y 231.318,Z 543.464,A -85,B 0,C 180,E1 -20577.624,E2 -20577.624} C_VEL
LIN {X 0,Y 228.48,Z 556.56,A -85,B 0,C 180,E1 -20579.38,E2 -20579.38} C_VEL
LIN {X 0,Y 225.426,Z 568.243,A -85,B 0,C 180,E1 -20581.359,E2 -20581.359} C_VEL
LIN {X 0,Y 222.904,Z 577.523,A -85,B 0,C 180,E1 -20583.303,E2 -20583.303} C_VEL
LIN {X 0,Y 219.902,Z 587.862,A -85,B 0,C 180,E1 -20585.954,E2 -20585.954} C_VEL
LIN {X 0,Y 217.402,Z 596.413,A -85,B 0,C 180,E1 -20588.674,E2 -20588.674} C_VEL
LIN {X 0,Y 215.17,Z 604.576,A -85,B 0,C 180,E1 -20591.924,E2 -20591.924} C_VEL
LIN {X 0,Y 213.667,Z 610.325,A -85,B 0,C 180,E1 -20594.744,E2 -20594.744} C_VEL
LIN {X 0,Y 212.255,Z 616.335,A -85,B 0,C 180,E1 -20598.541,E2 -20598.541} C_VEL
LIN {X 0,Y 211.612,Z 620.742,A -85,B 0,C 180,E1 -20602.366,E2 -20602.366} C_VEL
LIN {X 0,Y 211.435,Z 623.677,A -85,B 0,C 180,E1 -20606.188,E2 -20606.188} C_VEL
LIN {X 0,Y 211.563,Z 625.224,A -85,B 0,C 180,E1 -20610,E2 -20610} C_VEL
LIN {X 0,Y 211.395,Z 625.408,A -85,B 0,C 180,E1 -20613.812,E2 -20613.812} C_VEL
LIN {X 0,Y 211.619,Z 624.265,A -85,B 0,C 180,E1 -20617.634,E2 -20617.634} C_VEL
LIN {X 0,Y 212.382,Z 621.786,A -85,B 0,C 180,E1 -20621.452,E2 -20621.452} C_VEL
LIN {X 0,Y 213.937,Z 617.91,A -85,B 0,C 180,E1 -20625.236,E2 -20625.236} C_VEL
LIN {X 0,Y 216.296,Z 612.485,A -85,B 0,C 180,E1 -20628.961,E2 -20628.961} C_VEL
LIN {X 0,Y 218.509,Z 607.331,A -85,B 0,C 180,E1 -20631.708,E2 -20631.708} C_VEL
LIN {X 0,Y 221.812,Z 599.967,A -85,B 0,C 180,E1 -20634.822,E2 -20634.822} C_VEL
LIN {X 0,Y 225.753,Z 590.837,A -85,B 0,C 180,E1 -20637.837,E2 -20637.837} C_VEL
LIN {X 0,Y 229.726,Z 581.31,A -85,B 0,C 180,E1 -20640.316,E2 -20640.316} C_VEL
LIN {X 0,Y 233.44,Z 571.366,A -85,B 0,C 180,E1 -20642.415,E2 -20642.415} C_VEL
LIN {X 0,Y 237.103,Z 560.442,A -85,B 0,C 180,E1 -20644.275,E2 -20644.275} C_VEL
LIN {X 0,Y 240.833,Z 547.835,A -85,B 0,C 180,E1 -20645.964,E2 -20645.964} C_VEL
LIN {X 0,Y 243.945,Z 535.597,A -85,B 0,C 180,E1 -20647.228,E2 -20647.228} C_VEL
LIN {X 0,Y 246.731,Z 522.089,A -85,B 0,C 180,E1 -20648.281,E2 -20648.281} C_VEL
LIN {X 0,Y 248.842,Z 508.16,A -85,B 0,C 180,E1 -20649.061,E2 -20649.061} C_VEL
LIN {X 0,Y 250.191,Z 493.711,A -85,B 0,C 180,E1 -20649.59,E2 -20649.59} C_VEL
LIN {X 0,Y 253.692,Z 428.908,A -85,B 0,C 180,E1 -20651.329,E2 -20651.329} C_VEL
LIN {X 0,Y 246.506,Z 412.341,A -85,B 0,C 180,E1 -20653.632,E2 -20653.632} C_VEL
LIN {X 0,Y 239.448,Z 398.594,A -85,B 0,C 180,E1 -20656.025,E2 -20656.025} C_VEL
LIN {X 0,Y 232.746,Z 387.031,A -85,B 0,C 180,E1 -20658.483,E2 -20658.483} C_VEL
LIN {X 0,Y 228.712,Z 380.675,A -85,B 0,C 180,E1 -20660.071,E2 -20660.071} C_VEL
LIN {X 0,Y 226.14,Z 376.688,A -85,B 0,C 180,E1 -20661.143,E2 -20661.143} C_VEL
LIN {X 0,Y 222.441,Z 371.183,A -85,B 0,C 180,E1 -20662.766,E2 -20662.766} C_VEL
LIN {X 0,Y 218.357,Z 365.433,A -85,B 0,C 180,E1 -20664.689,E2 -20664.689} C_VEL
LIN {X 0,Y 215.351,Z 361.434,A -85,B 0,C 180,E1 -20666.206,E2 -20666.206} C_VEL
LIN {X 0,Y 214.59,Z 359.989,A -85,B 0,C 180,E1 -20666.731,E2 -20666.731} C_VEL
LIN {X 0,Y 213.748,Z 357.448,A -85,B 0,C 180,E1 -20668.914,E2 -20668.914} C_VEL
LIN {X 0,Y 213.78,Z 357.464,A -85,B 0,C 180,E1 -20672.597,E2 -20672.597} C_VEL
LIN {X 0,Y 213.805,Z 357.475,A -85,B 0,C 180,E1 -20676.98,E2 -20676.98} C_VEL
LIN {X 0,Y 213.886,Z 357.459,A -85,B 0,C 180,E1 -20682.799,E2 -20682.799} C_VEL
LIN {X 0,Y 213.927,Z 357.459,A -85,B 0,C 180,E1 -20686.706,E2 -20686.706} C_VEL
LIN {X 0,Y 214.121,Z 357.439,A -85,B 0,C 180,E1 -20690.555,E2 -20690.555} C_VEL
LIN {X 0,Y 214.066,Z 357.437,A -85,B 0,C 180,E1 -20694.348,E2 -20694.348} C_VEL
LIN {X 0,Y 214.398,Z 357.389,A -85,B 0,C 180,E1 -20698.122,E2 -20698.122} C_VEL
LIN {X 0,Y 214.503,Z 357.391,A -85,B 0,C 180,E1 -20700.001,E2 -20700.001} C_VEL
LIN {X 0,Y 214.401,Z 357.391,A -85,B 0,C 180,E1 -20701.879,E2 -20701.879} C_VEL
LIN {X 0,Y 214.18,Z 357.416,A -85,B 0,C 180,E1 -20707.543,E2 -20707.543} C_VEL
LIN {X 0,Y 213.986,Z 357.443,A -85,B 0,C 180,E1 -20711.366,E2 -20711.366} C_VEL
LIN {X 0,Y 213.892,Z 357.461,A -85,B 0,C 180,E1 -20715.241,E2 -20715.241} C_VEL
LIN {X 0,Y 213.795,Z 357.477,A -85,B 0,C 180,E1 -20719.192,E2 -20719.192} C_VEL
LIN {X 0,Y 213.806,Z 357.474,A -85,B 0,C 180,E1 -20723.233,E2 -20723.233} C_VEL
LIN {X 0,Y 213.836,Z 357.467,A -85,B 0,C 180,E1 -20727.258,E2 -20727.258} C_VEL
LIN {X 0,Y 214.701,Z 360.152,A -85,B 0,C 180,E1 -20727.86,E2 -20727.86} C_VEL
LIN {X 0,Y 216.656,Z 362.329,A -85,B 0,C 180,E1 -20728.851,E2 -20728.851} C_VEL
LIN {X 0,Y 218.079,Z 363.394,A -85,B 0,C 180,E1 -20729.513,E2 -20729.513} C_VEL
LIN {X 0,Y 219.867,Z 366.416,A -85,B 0,C 180,E1 -20730.413,E2 -20730.413} C_VEL
LIN {X 0,Y 222.221,Z 368.778,A -85,B 0,C 180,E1 -20731.454,E2 -20731.454} C_VEL
LIN {X 0,Y 224.66,Z 372.231,A -85,B 0,C 180,E1 -20732.538,E2 -20732.538} C_VEL
LIN {X 0,Y 226.149,Z 374.017,A -85,B 0,C 180,E1 -20733.157,E2 -20733.157} C_VEL
LIN {X 0,Y 229.771,Z 378.913,A -85,B 0,C 180,E1 -20734.622,E2 -20734.622} C_VEL
LIN {X 0,Y 235.268,Z 386.622,A -85,B 0,C 180,E1 -20736.688,E2 -20736.688} C_VEL
LIN {X 0,Y 241.645,Z 396.49,A -85,B 0,C 180,E1 -20738.906,E2 -20738.906} C_VEL
LIN {X 0,Y 248.025,Z 408.477,A -85,B 0,C 180,E1 -20741.011,E2 -20741.011} C_VEL
LIN {X 0,Y 253.758,Z 420.538,A -85,B 0,C 180,E1 -20742.8,E2 -20742.8} C_VEL
LIN {X 0,Y 254.152,Z 421.42,A -85,B 0,C 180,E1 -20742.92,E2 -20742.92} C_VEL
LIN {X 0,Y 250.178,Z 489.722,A -85,B 0,C 180,E1 -20744.754,E2 -20744.754} C_VEL
LIN {X 0,Y 248.535,Z 504.279,A -85,B 0,C 180,E1 -20745.443,E2 -20745.443} C_VEL
LIN {X 0,Y 246.166,Z 518.833,A -85,B 0,C 180,E1 -20746.469,E2 -20746.469} C_VEL
LIN {X 0,Y 243.557,Z 530.802,A -85,B 0,C 180,E1 -20747.586,E2 -20747.586} C_VEL
LIN {X 0,Y 240.147,Z 543.465,A -85,B 0,C 180,E1 -20749.096,E2 -20749.096} C_VEL
LIN {X 0,Y 236.681,Z 554.653,A -85,B 0,C 180,E1 -20750.801,E2 -20750.801} C_VEL
LIN {X 0,Y 232.69,Z 565.528,A -85,B 0,C 180,E1 -20752.84,E2 -20752.84} C_VEL
LIN {X 0,Y 228.715,Z 575.991,A -85,B 0,C 180,E1 -20755.357,E2 -20755.357} C_VEL
LIN {X 0,Y 225.186,Z 584.588,A -85,B 0,C 180,E1 -20757.957,E2 -20757.957} C_VEL
LIN {X 0,Y 221.476,Z 592.763,A -85,B 0,C 180,E1 -20761.059,E2 -20761.059} C_VEL
LIN {X 0,Y 218.329,Z 599.461,A -85,B 0,C 180,E1 -20764.334,E2 -20764.334} C_VEL
LIN {X 0,Y 215.579,Z 605.105,A -85,B 0,C 180,E1 -20767.982,E2 -20767.982} C_VEL
LIN {X 0,Y 214.016,Z 608.409,A -85,B 0,C 180,E1 -20770.83,E2 -20770.83} C_VEL
LIN {X 0,Y 212.523,Z 611.472,A -85,B 0,C 180,E1 -20774.66,E2 -20774.66} C_VEL
LIN {X 0,Y 211.616,Z 613.15,A -85,B 0,C 180,E1 -20778.506,E2 -20778.506} C_VEL
LIN {X 0,Y 211.382,Z 613.489,A -85,B 0,C 180,E1 -20782.358,E2 -20782.358} C_VEL
LIN {X 0,Y 211.51,Z 612.82,A -85,B 0,C 180,E1 -20785.451,E2 -20785.451} C_VEL
LIN {X 0,Y 211.567,Z 611.527,A -85,B 0,C 180,E1 -20788.096,E2 -20788.096} C_VEL
LIN {X 0,Y 211.986,Z 608.55,A -85,B 0,C 180,E1 -20791.9,E2 -20791.9} C_VEL
LIN {X 0,Y 212.893,Z 604.149,A -85,B 0,C 180,E1 -20795.683,E2 -20795.683} C_VEL
LIN {X 0,Y 214.094,Z 599.779,A -85,B 0,C 180,E1 -20798.495,E2 -20798.495} C_VEL
LIN {X 0,Y 216.033,Z 593.458,A -85,B 0,C 180,E1 -20801.731,E2 -20801.731} C_VEL
LIN {X 0,Y 218.405,Z 585.614,A -85,B 0,C 180,E1 -20804.917,E2 -20804.917} C_VEL
LIN {X 0,Y 220.746,Z 577.427,A -85,B 0,C 180,E1 -20807.605,E2 -20807.605} C_VEL
LIN {X 0,Y 223.643,Z 567.558,A -85,B 0,C 180,E1 -20810.222,E2 -20810.222} C_VEL
LIN {X 0,Y 226.645,Z 556.589,A -85,B 0,C 180,E1 -20812.564,E2 -20812.564} C_VEL
LIN {X 0,Y 229.641,Z 544.324,A -85,B 0,C 180,E1 -20814.644,E2 -20814.644} C_VEL
LIN {X 0,Y 232.212,Z 532.185,A -85,B 0,C 180,E1 -20816.271,E2 -20816.271} C_VEL
LIN {X 0,Y 234.631,Z 518.697,A -85,B 0,C 180,E1 -20817.663,E2 -20817.663} C_VEL
LIN {X 0,Y 236.6,Z 504.536,A -85,B 0,C 180,E1 -20818.739,E2 -20818.739} C_VEL
LIN {X 0,Y 237.854,Z 490.596,A -85,B 0,C 180,E1 -20819.481,E2 -20819.481} C_VEL
LIN {X 0,Y 239.236,Z 464.172,A -85,B 0,C 180,E1 -20820.283,E2 -20820.283} C_VEL
LIN {X 0,Y 241.595,Z 409.768,A -85,B 0,C 180,E1 -20821.831,E2 -20821.831} C_VEL
LIN {X 0,Y 235.036,Z 393.718,A -85,B 0,C 180,E1 -20823.574,E2 -20823.574} C_VEL
LIN {X 0,Y 231.108,Z 385.942,A -85,B 0,C 180,E1 -20824.614,E2 -20824.614} C_VEL
LIN {X 0,Y 222.942,Z 372.345,A -85,B 0,C 180,E1 -20826.839,E2 -20826.839} C_VEL
LIN {X 0,Y 218.65,Z 365.773,A -85,B 0,C 180,E1 -20828.082,E2 -20828.082} C_VEL
LIN {X 0,Y 216.186,Z 361.981,A -85,B 0,C 180,E1 -20828.83,E2 -20828.83} C_VEL
LIN {X 0,Y 214.34,Z 359.487,A -85,B 0,C 180,E1 -20829.391,E2 -20829.391} C_VEL
LIN {X 0,Y 213.773,Z 357.46,A -85,B 0,C 180,E1 -20829.693,E2 -20829.693} C_VEL
LIN {X 0,Y 213.703,Z 357.489,A -85,B 0,C 180,E1 -20833.678,E2 -20833.678} C_VEL
LIN {X 0,Y 213.702,Z 357.491,A -85,B 0,C 180,E1 -20836.343,E2 -20836.343} C_VEL
LIN {X 0,Y 213.715,Z 357.482,A -85,B 0,C 180,E1 -20839.142,E2 -20839.142} C_VEL
LIN {X 0,Y 213.742,Z 357.483,A -85,B 0,C 180,E1 -20843.71,E2 -20843.71} C_VEL
LIN {X 0,Y 213.778,Z 357.48,A -85,B 0,C 180,E1 -20848.73,E2 -20848.73} C_VEL
LIN {X 0,Y 213.823,Z 357.452,A -85,B 0,C 180,E1 -20852.602,E2 -20852.602} C_VEL
LIN {X 0,Y 213.796,Z 357.474,A -85,B 0,C 180,E1 -20856.985,E2 -20856.985} C_VEL
LIN {X 0,Y 213.88,Z 357.466,A -85,B 0,C 180,E1 -20862.798,E2 -20862.798} C_VEL
LIN {X 0,Y 213.917,Z 357.435,A -85,B 0,C 180,E1 -20866.704,E2 -20866.704} C_VEL
LIN {X 0,Y 214.13,Z 357.434,A -85,B 0,C 180,E1 -20870.554,E2 -20870.554} C_VEL
LIN {X 0,Y 214.074,Z 357.417,A -85,B 0,C 180,E1 -20874.347,E2 -20874.347} C_VEL
LIN {X 0,Y 214.399,Z 357.396,A -85,B 0,C 180,E1 -20878.121,E2 -20878.121} C_VEL
LIN {X 0,Y 214.501,Z 357.391,A -85,B 0,C 180,E1 -20879.999,E2 -20879.999} C_VEL
LIN {X 0,Y 214.368,Z 357.393,A -85,B 0,C 180,E1 -20881.878,E2 -20881.878} C_VEL
LIN {X 0,Y 214.168,Z 357.428,A -85,B 0,C 180,E1 -20887.542,E2 -20887.542} C_VEL
LIN {X 0,Y 213.981,Z 357.45,A -85,B 0,C 180,E1 -20891.365,E2 -20891.365} C_VEL
LIN {X 0,Y 213.895,Z 357.45,A -85,B 0,C 180,E1 -20895.239,E2 -20895.239} C_VEL
LIN {X 0,Y 213.806,Z 357.475,A -85,B 0,C 180,E1 -20899.19,E2 -20899.19} C_VEL
LIN {X 0,Y 213.796,Z 357.475,A -85,B 0,C 180,E1 -20903.232,E2 -20903.232} C_VEL
LIN {X 0,Y 213.781,Z 357.474,A -85,B 0,C 180,E1 -20907.428,E2 -20907.428} C_VEL
LIN {X 0,Y 213.732,Z 357.476,A -85,B 0,C 180,E1 -20910.551,E2 -20910.551} C_VEL
LIN {X 0,Y 213.099,Z 357.565,A -85,B 0,C 180,E1 -20912.123,E2 -20912.123} C_VEL
LIN {X 0,Y 210.279,Z 357.925,A -85,B 0,C 180,E1 -20914.691,E2 -20914.691} C_VEL
LIN {X 0,Y 207.009,Z 358.328,A -85,B 0,C 180,E1 -20917.868,E2 -20917.868} C_VEL
LIN {X 0,Y 206.66,Z 358.361,A -85,B 0,C 180,E1 -20918.97,E2 -20918.97} C_VEL
LIN {X 0,Y 206.68,Z 358.396,A -85,B 0,C 180,E1 -20920.984,E2 -20920.984} C_VEL
LIN {X 0,Y 207.495,Z 361.228,A -85,B 0,C 180,E1 -20922.551,E2 -20922.551} C_VEL
LIN {X 0,Y 210.113,Z 365.723,A -85,B 0,C 180,E1 -20923.457,E2 -20923.457} C_VEL
LIN {X 0,Y 216.45,Z 376.486,A -85,B 0,C 180,E1 -20925.504,E2 -20925.504} C_VEL
LIN {X 0,Y 223.972,Z 391.102,A -85,B 0,C 180,E1 -20927.787,E2 -20927.787} C_VEL
LIN {X 0,Y 231.009,Z 407.287,A -85,B 0,C 180,E1 -20929.826,E2 -20929.826} C_VEL
LIN {X 0,Y 234.521,Z 416.629,A -85,B 0,C 180,E1 -20930.827,E2 -20930.827} C_VEL
LIN {X 0,Y 235.339,Z 423.899,A -85,B 0,C 180,E1 -20931.242,E2 -20931.242} C_VEL
LIN {X 0,Y 231.632,Z 499.939,A -85,B 0,C 180,E1 -20933.457,E2 -20933.457} C_VEL
LIN {X 0,Y 230.106,Z 514.648,A -85,B 0,C 180,E1 -20934.193,E2 -20934.193} C_VEL
LIN {X 0,Y 228.031,Z 528.68,A -85,B 0,C 180,E1 -20935.239,E2 -20935.239} C_VEL
LIN {X 0,Y 225.335,Z 542.6,A -85,B 0,C 180,E1 -20936.654,E2 -20936.654} C_VEL
LIN {X 0,Y 222.534,Z 555.062,A -85,B 0,C 180,E1 -20938.327,E2 -20938.327} C_VEL
LIN {X 0,Y 219.558,Z 566.479,A -85,B 0,C 180,E1 -20940.255,E2 -20940.255} C_VEL
LIN {X 0,Y 216.524,Z 576.955,A -85,B 0,C 180,E1 -20942.45,E2 -20942.45} C_VEL
LIN {X 0,Y 213.385,Z 587.377,A -85,B 0,C 180,E1 -20945.171,E2 -20945.171} C_VEL
LIN {X 0,Y 210.753,Z 595.977,A -85,B 0,C 180,E1 -20947.967,E2 -20947.967} C_VEL
LIN {X 0,Y 208.318,Z 604.243,A -85,B 0,C 180,E1 -20951.337,E2 -20951.337} C_VEL
LIN {X 0,Y 206.778,Z 609.963,A -85,B 0,C 180,E1 -20954.223,E2 -20954.223} C_VEL
LIN {X 0,Y 205.512,Z 614.647,A -85,B 0,C 180,E1 -20957.157,E2 -20957.157} C_VEL
LIN {X 0,Y 204.668,Z 619.506,A -85,B 0,C 180,E1 -20961.111,E2 -20961.111} C_VEL
LIN {X 0,Y 204.388,Z 622.118,A -85,B 0,C 180,E1 -20964.079,E2 -20964.079} C_VEL
LIN {X 0,Y 204.366,Z 624.382,A -85,B 0,C 180,E1 -20968.029,E2 -20968.029} C_VEL
LIN {X 0,Y 204.48,Z 625.001,A -85,B 0,C 180,E1 -20970,E2 -20970} C_VEL
LIN {X 0,Y 204.295,Z 625.213,A -85,B 0,C 180,E1 -20973.945,E2 -20973.945} C_VEL
LIN {X 0,Y 204.555,Z 624.1,A -85,B 0,C 180,E1 -20977.899,E2 -20977.899} C_VEL
LIN {X 0,Y 205.39,Z 621.649,A -85,B 0,C 180,E1 -20981.847,E2 -20981.847} C_VEL
LIN {X 0,Y 207.053,Z 617.808,A -85,B 0,C 180,E1 -20985.756,E2 -20985.756} C_VEL
LIN {X 0,Y 209.531,Z 612.432,A -85,B 0,C 180,E1 -20989.597,E2 -20989.597} C_VEL
LIN {X 0,Y 211.882,Z 607.298,A -85,B 0,C 180,E1 -20992.423,E2 -20992.423} C_VEL
LIN {X 0,Y 215.356,Z 599.976,A -85,B 0,C 180,E1 -20995.619,E2 -20995.619} C_VEL
LIN {X 0,Y 219.492,Z 590.912,A -85,B 0,C 180,E1 -20998.703,E2 -20998.703} C_VEL
LIN {X 0,Y 223.625,Z 581.441,A -85,B 0,C 180,E1 -21001.234,E2 -21001.234} C_VEL
LIN {X 0,Y 227.467,Z 571.564,A -85,B 0,C 180,E1 -21003.376,E2 -21003.376} C_VEL
LIN {X 0,Y 231.295,Z 560.722,A -85,B 0,C 180,E1 -21005.261,E2 -21005.261} C_VEL
LIN {X 0,Y 235.148,Z 548.223,A -85,B 0,C 180,E1 -21006.975,E2 -21006.975} C_VEL
LIN {X 0,Y 238.351,Z 536.137,A -85,B 0,C 180,E1 -21008.257,E2 -21008.257} C_VEL
LIN {X 0,Y 241.236,Z 522.855,A -85,B 0,C 180,E1 -21009.319,E2 -21009.319} C_VEL
LIN {X 0,Y 243.534,Z 508.409,A -85,B 0,C 180,E1 -21010.15,E2 -21010.15} C_VEL
LIN {X 0,Y 244.924,Z 494.252,A -85,B 0,C 180,E1 -21010.684,E2 -21010.684} C_VEL
LIN {X 0,Y 248.546,Z 431.39,A -85,B 0,C 180,E1 -21012.378,E2 -21012.378} C_VEL
LIN {X 0,Y 242.014,Z 416.212,A -85,B 0,C 180,E1 -21014.584,E2 -21014.584} C_VEL
LIN {X 0,Y 235.433,Z 403.086,A -85,B 0,C 180,E1 -21016.937,E2 -21016.937} C_VEL
LIN {X 0,Y 229.193,Z 392.134,A -85,B 0,C 180,E1 -21019.34,E2 -21019.34} C_VEL
LIN {X 0,Y 223.3,Z 382.623,A -85,B 0,C 180,E1 -21021.824,E2 -21021.824} C_VEL
LIN {X 0,Y 219.262,Z 376.59,A -85,B 0,C 180,E1 -21023.672,E2 -21023.672} C_VEL
LIN {X 0,Y 215.676,Z 371.391,A -85,B 0,C 180,E1 -21025.444,E2 -21025.444} C_VEL
LIN {X 0,Y 212.591,Z 367.089,A -85,B 0,C 180,E1 -21027.085,E2 -21027.085} C_VEL
LIN {X 0,Y 211.822,Z 366.012,A -85,B 0,C 180,E1 -21027.515,E2 -21027.515} C_VEL
LIN {X 0,Y 207.359,Z 360.504,A -85,B 0,C 180,E1 -21030.146,E2 -21030.146} C_VEL
LIN {X 0,Y 206.982,Z 359.567,A -85,B 0,C 180,E1 -21030.506,E2 -21030.506} C_VEL
LIN {X 0,Y 206.698,Z 358.33,A -85,B 0,C 180,E1 -21031.759,E2 -21031.759} C_VEL
LIN {X 0,Y 206.739,Z 358.35,A -85,B 0,C 180,E1 -21036.61,E2 -21036.61} C_VEL
LIN {X 0,Y 206.82,Z 358.345,A -85,B 0,C 180,E1 -21042.192,E2 -21042.192} C_VEL
LIN {X 0,Y 206.869,Z 358.342,A -85,B 0,C 180,E1 -21046.243,E2 -21046.243} C_VEL
LIN {X 0,Y 207.067,Z 358.315,A -85,B 0,C 180,E1 -21050.23,E2 -21050.23} C_VEL
LIN {X 0,Y 207.029,Z 358.311,A -85,B 0,C 180,E1 -21054.155,E2 -21054.155} C_VEL
LIN {X 0,Y 207.338,Z 358.268,A -85,B 0,C 180,E1 -21058.058,E2 -21058.058} C_VEL
LIN {X 0,Y 207.472,Z 358.267,A -85,B 0,C 180,E1 -21060.001,E2 -21060.001} C_VEL
LIN {X 0,Y 207.341,Z 358.269,A -85,B 0,C 180,E1 -21061.943,E2 -21061.943} C_VEL
LIN {X 0,Y 207.124,Z 358.295,A -85,B 0,C 180,E1 -21067.801,E2 -21067.801} C_VEL
LIN {X 0,Y 206.909,Z 358.322,A -85,B 0,C 180,E1 -21071.76,E2 -21071.76} C_VEL
LIN {X 0,Y 206.819,Z 358.337,A -85,B 0,C 180,E1 -21075.775,E2 -21075.775} C_VEL
LIN {X 0,Y 206.716,Z 358.352,A -85,B 0,C 180,E1 -21079.877,E2 -21079.877} C_VEL
LIN {X 0,Y 206.743,Z 358.393,A -85,B 0,C 180,E1 -21083.798,E2 -21083.798} C_VEL
LIN {X 0,Y 207.489,Z 360.791,A -85,B 0,C 180,E1 -21084.382,E2 -21084.382} C_VEL
LIN {X 0,Y 209.302,Z 362.964,A -85,B 0,C 180,E1 -21085.482,E2 -21085.482} C_VEL
LIN {X 0,Y 211.282,Z 364.339,A -85,B 0,C 180,E1 -21086.552,E2 -21086.552} C_VEL
LIN {X 0,Y 212.937,Z 367.253,A -85,B 0,C 180,E1 -21087.522,E2 -21087.522} C_VEL
LIN {X 0,Y 215.508,Z 369.747,A -85,B 0,C 180,E1 -21088.819,E2 -21088.819} C_VEL
LIN {X 0,Y 217.962,Z 373.249,A -85,B 0,C 180,E1 -21090.053,E2 -21090.053} C_VEL
LIN {X 0,Y 219.591,Z 375.026,A -85,B 0,C 180,E1 -21090.803,E2 -21090.803} C_VEL
LIN {X 0,Y 222.319,Z 378.646,A -85,B 0,C 180,E1 -21092.04,E2 -21092.04} C_VEL
LIN {X 0,Y 227.309,Z 385.551,A -85,B 0,C 180,E1 -21094.151,E2 -21094.151} C_VEL
LIN {X 0,Y 232.2,Z 392.622,A -85,B 0,C 180,E1 -21096.057,E2 -21096.057} C_VEL
LIN {X 0,Y 237.769,Z 401.333,A -85,B 0,C 180,E1 -21098.075,E2 -21098.075} C_VEL
LIN {X 0,Y 244.375,Z 413.971,A -85,B 0,C 180,E1 -21100.351,E2 -21100.351} C_VEL
LIN {X 0,Y 248.936,Z 423.856,A -85,B 0,C 180,E1 -21101.847,E2 -21101.847} C_VEL
LIN {X 0,Y 245.013,Z 489.456,A -85,B 0,C 180,E1 -21103.63,E2 -21103.63} C_VEL
LIN {X 0,Y 243.366,Z 503.821,A -85,B 0,C 180,E1 -21104.306,E2 -21104.306} C_VEL
LIN {X 0,Y 240.995,Z 517.969,A -85,B 0,C 180,E1 -21105.29,E2 -21105.29} C_VEL
LIN {X 0,Y 238.294,Z 530.172,A -85,B 0,C 180,E1 -21106.419,E2 -21106.419} C_VEL
LIN {X 0,Y 234.757,Z 542.997,A -85,B 0,C 180,E1 -21107.946,E2 -21107.946} C_VEL
LIN {X 0,Y 230.795,Z 555.311,A -85,B 0,C 180,E1 -21109.842,E2 -21109.842} C_VEL
LIN {X 0,Y 226.972,Z 565.271,A -85,B 0,C 180,E1 -21111.738,E2 -21111.738} C_VEL
LIN {X 0,Y 222.828,Z 575.813,A -85,B 0,C 180,E1 -21114.305,E2 -21114.305} C_VEL
LIN {X 0,Y 219.054,Z 584.476,A -85,B 0,C 180,E1 -21116.948,E2 -21116.948} C_VEL
LIN {X 0,Y 215.173,Z 592.73,A -85,B 0,C 180,E1 -21120.127,E2 -21120.127} C_VEL
LIN {X 0,Y 211.961,Z 599.228,A -85,B 0,C 180,E1 -21123.342,E2 -21123.342} C_VEL
LIN {X 0,Y 208.902,Z 605.163,A -85,B 0,C 180,E1 -21127.24,E2 -21127.24} C_VEL
LIN {X 0,Y 207.199,Z 608.507,A -85,B 0,C 180,E1 -21130.173,E2 -21130.173} C_VEL
LIN {X 0,Y 205.596,Z 611.609,A -85,B 0,C 180,E1 -21134.13,E2 -21134.13} C_VEL
LIN {X 0,Y 204.576,Z 613.326,A -85,B 0,C 180,E1 -21138.105,E2 -21138.105} C_VEL
LIN {X 0,Y 204.284,Z 613.702,A -85,B 0,C 180,E1 -21142.09,E2 -21142.09} C_VEL
LIN {X 0,Y 204.414,Z 612.938,A -85,B 0,C 180,E1 -21145.613,E2 -21145.613} C_VEL
LIN {X 0,Y 204.463,Z 611.795,A -85,B 0,C 180,E1 -21148.03,E2 -21148.03} C_VEL
LIN {X 0,Y 204.92,Z 608.855,A -85,B 0,C 180,E1 -21151.965,E2 -21151.965} C_VEL
LIN {X 0,Y 205.861,Z 604.495,A -85,B 0,C 180,E1 -21155.878,E2 -21155.878} C_VEL
LIN {X 0,Y 207.583,Z 598.555,A -85,B 0,C 180,E1 -21159.746,E2 -21159.746} C_VEL
LIN {X 0,Y 209.766,Z 591.865,A -85,B 0,C 180,E1 -21163.07,E2 -21163.07} C_VEL
LIN {X 0,Y 212.191,Z 584.104,A -85,B 0,C 180,E1 -21166.152,E2 -21166.152} C_VEL
LIN {X 0,Y 214.483,Z 576.501,A -85,B 0,C 180,E1 -21168.631,E2 -21168.631} C_VEL
LIN {X 0,Y 217.586,Z 566.375,A -85,B 0,C 180,E1 -21171.307,E2 -21171.307} C_VEL
LIN {X 0,Y 220.767,Z 555.039,A -85,B 0,C 180,E1 -21173.697,E2 -21173.697} C_VEL
LIN {X 0,Y 223.572,Z 543.769,A -85,B 0,C 180,E1 -21175.609,E2 -21175.609} C_VEL
LIN {X 0,Y 226.224,Z 531.454,A -85,B 0,C 180,E1 -21177.272,E2 -21177.272} C_VEL
LIN {X 0,Y 228.777,Z 517.698,A -85,B 0,C 180,E1 -21178.684,E2 -21178.684} C_VEL
LIN {X 0,Y 230.732,Z 503.874,A -85,B 0,C 180,E1 -21179.729,E2 -21179.729} C_VEL
LIN {X 0,Y 232.068,Z 489.497,A -85,B 0,C 180,E1 -21180.481,E2 -21180.481} C_VEL
LIN {X 0,Y 235.775,Z 411.74,A -85,B 0,C 180,E1 -21182.767,E2 -21182.767} C_VEL
LIN {X 0,Y 229.67,Z 396.802,A -85,B 0,C 180,E1 -21184.472,E2 -21184.472} C_VEL
LIN {X 0,Y 226.028,Z 389.61,A -85,B 0,C 180,E1 -21185.483,E2 -21185.483} C_VEL
LIN {X 0,Y 217.373,Z 375.012,A -85,B 0,C 180,E1 -21187.981,E2 -21187.981} C_VEL
LIN {X 0,Y 211.74,Z 366.756,A -85,B 0,C 180,E1 -21189.714,E2 -21189.714} C_VEL
LIN {X 0,Y 209.401,Z 363.092,A -85,B 0,C 180,E1 -21190.488,E2 -21190.488} C_VEL
LIN {X 0,Y 207.498,Z 360.858,A -85,B 0,C 180,E1 -21191.102,E2 -21191.102} C_VEL
LIN {X 0,Y 206.654,Z 358.349,A -85,B 0,C 180,E1 -21191.492,E2 -21191.492} C_VEL
LIN {X 0,Y 206.63,Z 358.366,A -85,B 0,C 180,E1 -21195.581,E2 -21195.581} C_VEL
LIN {X 0,Y 206.658,Z 358.366,A -85,B 0,C 180,E1 -21199.747,E2 -21199.747} C_VEL
LIN {X 0,Y 206.697,Z 358.364,A -85,B 0,C 180,E1 -21204.687,E2 -21204.687} C_VEL
LIN {X 0,Y 206.704,Z 358.363,A -85,B 0,C 180,E1 -21209.335,E2 -21209.335} C_VEL
LIN {X 0,Y 206.726,Z 358.341,A -85,B 0,C 180,E1 -21213.77,E2 -21213.77} C_VEL
LIN {X 0,Y 206.712,Z 358.344,A -85,B 0,C 180,E1 -21218.037,E2 -21218.037} C_VEL
LIN {X 0,Y 206.817,Z 358.343,A -85,B 0,C 180,E1 -21222.191,E2 -21222.191} C_VEL
LIN {X 0,Y 206.858,Z 358.317,A -85,B 0,C 180,E1 -21226.241,E2 -21226.241} C_VEL
LIN {X 0,Y 207.074,Z 358.311,A -85,B 0,C 180,E1 -21230.229,E2 -21230.229} C_VEL
LIN {X 0,Y 207.037,Z 358.295,A -85,B 0,C 180,E1 -21234.154,E2 -21234.154} C_VEL
LIN {X 0,Y 207.339,Z 358.275,A -85,B 0,C 180,E1 -21238.057,E2 -21238.057} C_VEL
LIN {X 0,Y 207.468,Z 358.267,A -85,B 0,C 180,E1 -21239.999,E2 -21239.999} C_VEL
LIN {X 0,Y 207.012,Z 358.306,A -85,B 0,C 180,E1 -21243.893,E2 -21243.893} C_VEL
LIN {X 0,Y 207.113,Z 358.303,A -85,B 0,C 180,E1 -21247.8,E2 -21247.8} C_VEL
LIN {X 0,Y 206.905,Z 358.334,A -85,B 0,C 180,E1 -21251.759,E2 -21251.759} C_VEL
LIN {X 0,Y 206.823,Z 358.33,A -85,B 0,C 180,E1 -21255.774,E2 -21255.774} C_VEL
LIN {X 0,Y 206.725,Z 358.348,A -85,B 0,C 180,E1 -21259.874,E2 -21259.874} C_VEL
LIN {X 0,Y 206.732,Z 358.356,A -85,B 0,C 180,E1 -21264.075,E2 -21264.075} C_VEL
LIN {X 0,Y 206.683,Z 358.363,A -85,B 0,C 180,E1 -21268.427,E2 -21268.427} C_VEL
LIN {X 0,Y 206.69,Z 358.362,A -85,B 0,C 180,E1 -21272.959,E2 -21272.959} C_VEL
LIN {X 0,Y 206.676,Z 358.36,A -85,B 0,C 180,E1 -21277.74,E2 -21277.74} C_VEL
LIN {X 0,Y 206.66,Z 358.361,A -85,B 0,C 180,E1 -21278.97,E2 -21278.97} C_VEL
LIN {X 0,Y 206.725,Z 359.114,A -85,B 0,C 180,E1 -21279.995,E2 -21279.995} C_VEL
LIN {X 0,Y 206.974,Z 360.977,A -85,B 0,C 180,E1 -21280.916,E2 -21280.916} C_VEL
LIN {X 0,Y 207.631,Z 365.071,A -85,B 0,C 180,E1 -21282.082,E2 -21282.082} C_VEL
LIN {X 0,Y 208.65,Z 370.239,A -85,B 0,C 180,E1 -21283.032,E2 -21283.032} C_VEL
LIN {X 0,Y 209.546,Z 373.942,A -85,B 0,C 180,E1 -21283.595,E2 -21283.595} C_VEL
LIN {X 0,Y 212.104,Z 381.194,A -85,B 0,C 180,E1 -21284.666,E2 -21284.666} C_VEL
LIN {X 0,Y 218.932,Z 394.68,A -85,B 0,C 180,E1 -21286.85,E2 -21286.85} C_VEL
LIN {X 0,Y 225.547,Z 409.939,A -85,B 0,C 180,E1 -21288.867,E2 -21288.867} C_VEL
LIN {X 0,Y 229,Z 419.263,A -85,B 0,C 180,E1 -21289.907,E2 -21289.907} C_VEL
LIN {X 0,Y 229.588,Z 425.631,A -85,B 0,C 180,E1 -21290.262,E2 -21290.262} C_VEL
LIN {X 0,Y 225.737,Z 500.321,A -85,B 0,C 180,E1 -21292.48,E2 -21292.48} C_VEL
LIN {X 0,Y 224.138,Z 514.831,A -85,B 0,C 180,E1 -21293.225,E2 -21293.225} C_VEL
LIN {X 0,Y 221.997,Z 528.764,A -85,B 0,C 180,E1 -21294.29,E2 -21294.29} C_VEL
LIN {X 0,Y 219.398,Z 541.731,A -85,B 0,C 180,E1 -21295.628,E2 -21295.628} C_VEL
LIN {X 0,Y 216.355,Z 554.767,A -85,B 0,C 180,E1 -21297.398,E2 -21297.398} C_VEL
LIN {X 0,Y 213.05,Z 567.016,A -85,B 0,C 180,E1 -21299.525,E2 -21299.525} C_VEL
LIN {X 0,Y 210.22,Z 576.386,A -85,B 0,C 180,E1 -21301.55,E2 -21301.55} C_VEL
LIN {X 0,Y 206.9,Z 586.876,A -85,B 0,C 180,E1 -21304.337,E2 -21304.337} C_VEL
LIN {X 0,Y 204.122,Z 595.527,A -85,B 0,C 180,E1 -21307.212,E2 -21307.212} C_VEL
LIN {X 0,Y 201.674,Z 603.261,A -85,B 0,C 180,E1 -21310.4,E2 -21310.4} C_VEL
LIN {X 0,Y 199.908,Z 609.593,A -85,B 0,C 180,E1 -21313.666,E2 -21313.666} C_VEL
LIN {X 0,Y 198.543,Z 614.311,A -85,B 0,C 180,E1 -21316.698,E2 -21316.698} C_VEL
LIN {X 0,Y 197.625,Z 619.205,A -85,B 0,C 180,E1 -21320.792,E2 -21320.792} C_VEL
LIN {X 0,Y 197.302,Z 621.848,A -85,B 0,C 180,E1 -21323.866,E2 -21323.866} C_VEL
LIN {X 0,Y 197.271,Z 624.144,A -85,B 0,C 180,E1 -21327.958,E2 -21327.958} C_VEL
LIN {X 0,Y 197.379,Z 624.777,A -85,B 0,C 180,E1 -21330,E2 -21330} C_VEL
LIN {X 0,Y 197.204,Z 625.018,A -85,B 0,C 180,E1 -21334.087,E2 -21334.087} C_VEL
LIN {X 0,Y 197.492,Z 623.934,A -85,B 0,C 180,E1 -21338.183,E2 -21338.183} C_VEL
LIN {X 0,Y 198.416,Z 621.515,A -85,B 0,C 180,E1 -21342.27,E2 -21342.27} C_VEL
LIN {X 0,Y 200.193,Z 617.705,A -85,B 0,C 180,E1 -21346.31,E2 -21346.31} C_VEL
LIN {X 0,Y 202.796,Z 612.379,A -85,B 0,C 180,E1 -21350.276,E2 -21350.276} C_VEL
LIN {X 0,Y 205.3,Z 607.264,A -85,B 0,C 180,E1 -21353.183,E2 -21353.183} C_VEL
LIN {X 0,Y 208.959,Z 599.983,A -85,B 0,C 180,E1 -21356.464,E2 -21356.464} C_VEL
LIN {X 0,Y 213.279,Z 590.988,A -85,B 0,C 180,E1 -21359.622,E2 -21359.622} C_VEL
LIN {X 0,Y 217.588,Z 581.572,A -85,B 0,C 180,E1 -21362.204,E2 -21362.204} C_VEL
LIN {X 0,Y 221.914,Z 570.805,A -85,B 0,C 180,E1 -21364.572,E2 -21364.572} C_VEL
LIN {X 0,Y 225.969,Z 559.716,A -85,B 0,C 180,E1 -21366.499,E2 -21366.499} C_VEL
LIN {X 0,Y 229.543,Z 548.611,A -85,B 0,C 180,E1 -21368.036,E2 -21368.036} C_VEL
LIN {X 0,Y 232.844,Z 536.679,A -85,B 0,C 180,E1 -21369.333,E2 -21369.333} C_VEL
LIN {X 0,Y 235.822,Z 523.625,A -85,B 0,C 180,E1 -21370.404,E2 -21370.404} C_VEL
LIN {X 0,Y 238.178,Z 509.579,A -85,B 0,C 180,E1 -21371.246,E2 -21371.246} C_VEL
LIN {X 0,Y 239.743,Z 494.813,A -85,B 0,C 180,E1 -21371.828,E2 -21371.828} C_VEL
LIN {X 0,Y 243.418,Z 433.742,A -85,B 0,C 180,E1 -21373.494,E2 -21373.494} C_VEL
LIN {X 0,Y 237.443,Z 419.652,A -85,B 0,C 180,E1 -21375.631,E2 -21375.631} C_VEL
LIN {X 0,Y 230.761,Z 406.284,A -85,B 0,C 180,E1 -21378.158,E2 -21378.158} C_VEL
LIN {X 0,Y 223.723,Z 393.758,A -85,B 0,C 180,E1 -21381.077,E2 -21381.077} C_VEL
LIN {X 0,Y 217.074,Z 383.222,A -85,B 0,C 180,E1 -21384.152,E2 -21384.152} C_VEL
LIN {X 0,Y 212.901,Z 377.166,A -85,B 0,C 180,E1 -21386.29,E2 -21386.29} C_VEL
LIN {X 0,Y 209.19,Z 371.951,A -85,B 0,C 180,E1 -21388.38,E2 -21388.38} C_VEL
LIN {X 0,Y 204.943,Z 366.4,A -85,B 0,C 180,E1 -21391.029,E2 -21391.029} C_VEL
LIN {X 0,Y 203.704,Z 364.771,A -85,B 0,C 180,E1 -21391.872,E2 -21391.872} C_VEL
LIN {X 0,Y 201.225,Z 362.878,A -85,B 0,C 180,E1 -21393.558,E2 -21393.558} C_VEL
LIN {X 0,Y 199.923,Z 360.521,A -85,B 0,C 180,E1 -21394.632,E2 -21394.632} C_VEL
LIN {X 0,Y 199.645,Z 359.23,A -85,B 0,C 180,E1 -21395.012,E2 -21395.012} C_VEL
LIN {X 0,Y 199.656,Z 359.227,A -85,B 0,C 180,E1 -21399.391,E2 -21399.391} C_VEL
LIN {X 0,Y 199.76,Z 359.213,A -85,B 0,C 180,E1 -21403.653,E2 -21403.653} C_VEL
LIN {X 0,Y 199.856,Z 359.201,A -85,B 0,C 180,E1 -21407.82,E2 -21407.82} C_VEL
LIN {X 0,Y 200.063,Z 359.179,A -85,B 0,C 180,E1 -21411.923,E2 -21411.923} C_VEL
LIN {X 0,Y 200.28,Z 359.146,A -85,B 0,C 180,E1 -21417.99,E2 -21417.99} C_VEL
LIN {X 0,Y 200.439,Z 359.142,A -85,B 0,C 180,E1 -21420.001,E2 -21420.001} C_VEL
LIN {X 0,Y 199.991,Z 359.189,A -85,B 0,C 180,E1 -21424.031,E2 -21424.031} C_VEL
LIN {X 0,Y 200.071,Z 359.174,A -85,B 0,C 180,E1 -21428.078,E2 -21428.078} C_VEL
LIN {X 0,Y 199.858,Z 359.2,A -85,B 0,C 180,E1 -21432.181,E2 -21432.181} C_VEL
LIN {X 0,Y 199.757,Z 359.214,A -85,B 0,C 180,E1 -21436.348,E2 -21436.348} C_VEL
LIN {X 0,Y 199.695,Z 359.269,A -85,B 0,C 180,E1 -21439.533,E2 -21439.533} C_VEL
LIN {X 0,Y 200.37,Z 361.535,A -85,B 0,C 180,E1 -21440.199,E2 -21440.199} C_VEL
LIN {X 0,Y 201.988,Z 363.635,A -85,B 0,C 180,E1 -21441.429,E2 -21441.429} C_VEL
LIN {X 0,Y 204.503,Z 365.377,A -85,B 0,C 180,E1 -21443.078,E2 -21443.078} C_VEL
LIN {X 0,Y 206.147,Z 368.265,A -85,B 0,C 180,E1 -21444.216,E2 -21444.216} C_VEL
LIN {X 0,Y 208.957,Z 370.815,A -85,B 0,C 180,E1 -21445.862,E2 -21445.862} C_VEL
LIN {X 0,Y 211.085,Z 374.051,A -85,B 0,C 180,E1 -21447.112,E2 -21447.112} C_VEL
LIN {X 0,Y 213.069,Z 376.097,A -85,B 0,C 180,E1 -21448.153,E2 -21448.153} C_VEL
LIN {X 0,Y 216.037,Z 380.016,A -85,B 0,C 180,E1 -21449.671,E2 -21449.671} C_VEL
LIN {X 0,Y 220.879,Z 386.543,A -85,B 0,C 180,E1 -21451.946,E2 -21451.946} C_VEL
LIN {X 0,Y 225.84,Z 393.446,A -85,B 0,C 180,E1 -21454.067,E2 -21454.067} C_VEL
LIN {X 0,Y 233.274,Z 404.972,A -85,B 0,C 180,E1 -21456.965,E2 -21456.965} C_VEL
LIN {X 0,Y 238.87,Z 415.674,A -85,B 0,C 180,E1 -21459.012,E2 -21459.012} C_VEL
LIN {X 0,Y 243.831,Z 426.24,A -85,B 0,C 180,E1 -21460.73,E2 -21460.73} C_VEL
LIN {X 0,Y 239.924,Z 489.334,A -85,B 0,C 180,E1 -21462.463,E2 -21462.463} C_VEL
LIN {X 0,Y 238.286,Z 503.371,A -85,B 0,C 180,E1 -21463.117,E2 -21463.117} C_VEL
LIN {X 0,Y 235.942,Z 517.114,A -85,B 0,C 180,E1 -21464.062,E2 -21464.062} C_VEL
LIN {X 0,Y 233.127,Z 529.544,A -85,B 0,C 180,E1 -21465.198,E2 -21465.198} C_VEL
LIN {X 0,Y 229.488,Z 542.531,A -85,B 0,C 180,E1 -21466.748,E2 -21466.748} C_VEL
LIN {X 0,Y 225.542,Z 554.278,A -85,B 0,C 180,E1 -21468.536,E2 -21468.536} C_VEL
LIN {X 0,Y 221.358,Z 565.014,A -85,B 0,C 180,E1 -21470.582,E2 -21470.582} C_VEL
LIN {X 0,Y 216.998,Z 575.633,A -85,B 0,C 180,E1 -21473.191,E2 -21473.191} C_VEL
LIN {X 0,Y 213.024,Z 584.36,A -85,B 0,C 180,E1 -21475.886,E2 -21475.886} C_VEL
LIN {X 0,Y 208.938,Z 592.693,A -85,B 0,C 180,E1 -21479.14,E2 -21479.14} C_VEL
LIN {X 0,Y 205.382,Z 599.482,A -85,B 0,C 180,E1 -21482.58,E2 -21482.58} C_VEL
LIN {X 0,Y 202.233,Z 605.221,A -85,B 0,C 180,E1 -21486.444,E2 -21486.444} C_VEL
LIN {X 0,Y 200.404,Z 608.602,A -85,B 0,C 180,E1 -21489.471,E2 -21489.471} C_VEL
LIN {X 0,Y 198.686,Z 611.747,A -85,B 0,C 180,E1 -21493.562,E2 -21493.562} C_VEL
LIN {X 0,Y 197.546,Z 613.501,A -85,B 0,C 180,E1 -21497.675,E2 -21497.675} C_VEL
LIN {X 0,Y 197.208,Z 613.914,A -85,B 0,C 180,E1 -21501.805,E2 -21501.805} C_VEL
LIN {X 0,Y 197.328,Z 613.006,A -85,B 0,C 180,E1 -21505.915,E2 -21505.915} C_VEL
LIN {X 0,Y 197.556,Z 610.782,A -85,B 0,C 180,E1 -21510,E2 -21510} C_VEL
LIN {X 0,Y 198.238,Z 607.185,A -85,B 0,C 180,E1 -21514.066,E2 -21514.066} C_VEL
LIN {X 0,Y 199.624,Z 602.102,A -85,B 0,C 180,E1 -21518.095,E2 -21518.095} C_VEL
LIN {X 0,Y 201.196,Z 597.171,A -85,B 0,C 180,E1 -21521.076,E2 -21521.076} C_VEL
LIN {X 0,Y 203.618,Z 590.067,A -85,B 0,C 180,E1 -21524.511,E2 -21524.511} C_VEL
LIN {X 0,Y 205.958,Z 582.741,A -85,B 0,C 180,E1 -21527.371,E2 -21527.371} C_VEL
LIN {X 0,Y 208.815,Z 573.884,A -85,B 0,C 180,E1 -21530.18,E2 -21530.18} C_VEL
LIN {X 0,Y 212.194,Z 563.154,A -85,B 0,C 180,E1 -21532.902,E2 -21532.902} C_VEL
LIN {X 0,Y 215.284,Z 552.286,A -85,B 0,C 180,E1 -21535.111,E2 -21535.111} C_VEL
LIN {X 0,Y 218.28,Z 540.38,A -85,B 0,C 180,E1 -21537.05,E2 -21537.05} C_VEL
LIN {X 0,Y 221.131,Z 527.138,A -85,B 0,C 180,E1 -21538.73,E2 -21538.73} C_VEL
LIN {X 0,Y 223.418,Z 514.342,A -85,B 0,C 180,E1 -21539.958,E2 -21539.958} C_VEL
LIN {X 0,Y 225.194,Z 500.705,A -85,B 0,C 180,E1 -21540.927,E2 -21540.927} C_VEL
LIN {X 0,Y 226.43,Z 486.761,A -85,B 0,C 180,E1 -21541.585,E2 -21541.585} C_VEL
LIN {X 0,Y 230.005,Z 413.605,A -85,B 0,C 180,E1 -21543.758,E2 -21543.758} C_VEL
LIN {X 0,Y 223.888,Z 398.796,A -85,B 0,C 180,E1 -21545.555,E2 -21545.555} C_VEL
LIN {X 0,Y 218.347,Z 388.706,A -85,B 0,C 180,E1 -21547.171,E2 -21547.171} C_VEL
LIN {X 0,Y 212.468,Z 378.96,A -85,B 0,C 180,E1 -21548.98,E2 -21548.98} C_VEL
LIN {X 0,Y 207.396,Z 371.402,A -85,B 0,C 180,E1 -21550.629,E2 -21550.629} C_VEL
LIN {X 0,Y 205.085,Z 368.01,A -85,B 0,C 180,E1 -21551.422,E2 -21551.422} C_VEL
LIN {X 0,Y 202.935,Z 364.777,A -85,B 0,C 180,E1 -21552.189,E2 -21552.189} C_VEL
LIN {X 0,Y 200.313,Z 361.634,A -85,B 0,C 180,E1 -21553.121,E2 -21553.121} C_VEL
LIN {X 0,Y 199.567,Z 359.251,A -85,B 0,C 180,E1 -21553.512,E2 -21553.512} C_VEL
LIN {X 0,Y 199.577,Z 359.242,A -85,B 0,C 180,E1 -21558.003,E2 -21558.003} C_VEL
LIN {X 0,Y 199.609,Z 359.245,A -85,B 0,C 180,E1 -21560.766,E2 -21560.766} C_VEL
LIN {X 0,Y 199.609,Z 359.238,A -85,B 0,C 180,E1 -21565.712,E2 -21565.712} C_VEL
LIN {X 0,Y 199.69,Z 359.231,A -85,B 0,C 180,E1 -21568.134,E2 -21568.134} C_VEL
LIN {X 0,Y 199.681,Z 359.213,A -85,B 0,C 180,E1 -21572.77,E2 -21572.77} C_VEL
LIN {X 0,Y 199.675,Z 359.231,A -85,B 0,C 180,E1 -21577.221,E2 -21577.221} C_VEL
LIN {X 0,Y 199.741,Z 359.217,A -85,B 0,C 180,E1 -21581.802,E2 -21581.802} C_VEL
LIN {X 0,Y 199.796,Z 359.201,A -85,B 0,C 180,E1 -21585.745,E2 -21585.745} C_VEL
LIN {X 0,Y 200.018,Z 359.185,A -85,B 0,C 180,E1 -21589.881,E2 -21589.881} C_VEL
LIN {X 0,Y 200,Z 359.173,A -85,B 0,C 180,E1 -21593.948,E2 -21593.948} C_VEL
LIN {X 0,Y 200.281,Z 359.151,A -85,B 0,C 180,E1 -21597.988,E2 -21597.988} C_VEL
LIN {X 0,Y 200.435,Z 359.144,A -85,B 0,C 180,E1 -21599.999,E2 -21599.999} C_VEL
LIN {X 0,Y 199.96,Z 359.185,A -85,B 0,C 180,E1 -21604.03,E2 -21604.03} C_VEL
LIN {X 0,Y 200.062,Z 359.177,A -85,B 0,C 180,E1 -21608.077,E2 -21608.077} C_VEL
LIN {X 0,Y 199.856,Z 359.214,A -85,B 0,C 180,E1 -21612.18,E2 -21612.18} C_VEL
LIN {X 0,Y 199.76,Z 359.211,A -85,B 0,C 180,E1 -21616.347,E2 -21616.347} C_VEL
LIN {X 0,Y 199.655,Z 359.223,A -85,B 0,C 180,E1 -21620.609,E2 -21620.609} C_VEL
LIN {X 0,Y 199.644,Z 359.231,A -85,B 0,C 180,E1 -21624.988,E2 -21624.988} C_VEL
LIN {X 0,Y 199.603,Z 359.238,A -85,B 0,C 180,E1 -21629.533,E2 -21629.533} C_VEL
LIN {X 0,Y 199.66,Z 359.24,A -85,B 0,C 180,E1 -21632.353,E2 -21632.353} C_VEL
LIN {X 0,Y 199.619,Z 359.241,A -85,B 0,C 180,E1 -21636.763,E2 -21636.763} C_VEL
LIN {X 0,Y 199.638,Z 359.326,A -85,B 0,C 180,E1 -21639.484,E2 -21639.484} C_VEL
LIN {X 0,Y 200.126,Z 361.119,A -85,B 0,C 180,E1 -21640.434,E2 -21640.434} C_VEL
LIN {X 0,Y 203.06,Z 365.69,A -85,B 0,C 180,E1 -21641.53,E2 -21641.53} C_VEL
LIN {X 0,Y 210.446,Z 378.289,A -85,B 0,C 180,E1 -21644.12,E2 -21644.12} C_VEL
LIN {X 0,Y 212.104,Z 381.194,A -85,B 0,C 180,E1 -21644.666,E2 -21644.666} C_VEL
LIN {X 0,Y 213.946,Z 386.227,A -85,B 0,C 180,E1 -21645.338,E2 -21645.338} C_VEL
LIN {X 0,Y 215.92,Z 395.375,A -85,B 0,C 180,E1 -21646.2,E2 -21646.2} C_VEL
LIN {X 0,Y 218.093,Z 406.567,A -85,B 0,C 180,E1 -21647.166,E2 -21647.166} C_VEL
LIN {X 0,Y 219.155,Z 410.12,A -85,B 0,C 180,E1 -21647.546,E2 -21647.546} C_VEL
LIN {X 0,Y 223.513,Z 421.909,A -85,B 0,C 180,E1 -21648.936,E2 -21648.936} C_VEL
LIN {X 0,Y 223.913,Z 426.83,A -85,B 0,C 180,E1 -21649.213,E2 -21649.213} C_VEL
LIN {X 0,Y 219.995,Z 499.54,A -85,B 0,C 180,E1 -21651.396,E2 -21651.396} C_VEL
LIN {X 0,Y 218.342,Z 514.244,A -85,B 0,C 180,E1 -21652.152,E2 -21652.152} C_VEL
LIN {X 0,Y 216.238,Z 527.71,A -85,B 0,C 180,E1 -21653.186,E2 -21653.186} C_VEL
LIN {X 0,Y 213.521,Z 540.861,A -85,B 0,C 180,E1 -21654.542,E2 -21654.542} C_VEL
LIN {X 0,Y 210.482,Z 553.6,A -85,B 0,C 180,E1 -21656.284,E2 -21656.284} C_VEL
LIN {X 0,Y 207.256,Z 565.322,A -85,B 0,C 180,E1 -21658.324,E2 -21658.324} C_VEL
LIN {X 0,Y 203.982,Z 575.817,A -85,B 0,C 180,E1 -21660.597,E2 -21660.597} C_VEL
LIN {X 0,Y 200.436,Z 586.364,A -85,B 0,C 180,E1 -21663.446,E2 -21663.446} C_VEL
LIN {X 0,Y 197.529,Z 595.069,A -85,B 0,C 180,E1 -21666.406,E2 -21666.406} C_VEL
LIN {X 0,Y 194.732,Z 603.438,A -85,B 0,C 180,E1 -21669.973,E2 -21669.973} C_VEL
LIN {X 0,Y 193.027,Z 609.218,A -85,B 0,C 180,E1 -21673.066,E2 -21673.066} C_VEL
LIN {X 0,Y 191.6,Z 613.975,A -85,B 0,C 180,E1 -21676.207,E2 -21676.207} C_VEL
LIN {X 0,Y 190.567,Z 618.902,A -85,B 0,C 180,E1 -21680.447,E2 -21680.447} C_VEL
LIN {X 0,Y 190.218,Z 621.578,A -85,B 0,C 180,E1 -21683.636,E2 -21683.636} C_VEL
LIN {X 0,Y 190.179,Z 623.905,A -85,B 0,C 180,E1 -21687.882,E2 -21687.882} C_VEL
LIN {X 0,Y 190.281,Z 624.553,A -85,B 0,C 180,E1 -21690,E2 -21690} C_VEL
LIN {X 0,Y 190.125,Z 624.824,A -85,B 0,C 180,E1 -21694.24,E2 -21694.24} C_VEL
LIN {X 0,Y 190.451,Z 623.769,A -85,B 0,C 180,E1 -21698.488,E2 -21698.488} C_VEL
LIN {X 0,Y 191.441,Z 621.38,A -85,B 0,C 180,E1 -21702.724,E2 -21702.724} C_VEL
LIN {X 0,Y 193.356,Z 617.602,A -85,B 0,C 180,E1 -21706.904,E2 -21706.904} C_VEL
LIN {X 0,Y 196.092,Z 612.322,A -85,B 0,C 180,E1 -21711.002,E2 -21711.002} C_VEL
LIN {X 0,Y 198.76,Z 607.231,A -85,B 0,C 180,E1 -21713.993,E2 -21713.993} C_VEL
LIN {X 0,Y 202.609,Z 599.989,A -85,B 0,C 180,E1 -21717.361,E2 -21717.361} C_VEL
LIN {X 0,Y 207.126,Z 591.058,A -85,B 0,C 180,E1 -21720.594,E2 -21720.594} C_VEL
LIN {X 0,Y 211.617,Z 581.705,A -85,B 0,C 180,E1 -21723.227,E2 -21723.227} C_VEL
LIN {X 0,Y 215.861,Z 571.639,A -85,B 0,C 180,E1 -21725.517,E2 -21725.517} C_VEL
LIN {X 0,Y 220.322,Z 560.003,A -85,B 0,C 180,E1 -21727.593,E2 -21727.593} C_VEL
LIN {X 0,Y 224.019,Z 549.009,A -85,B 0,C 180,E1 -21729.15,E2 -21729.15} C_VEL
LIN {X 0,Y 227.422,Z 537.232,A -85,B 0,C 180,E1 -21730.462,E2 -21730.462} C_VEL
LIN {X 0,Y 230.488,Z 524.41,A -85,B 0,C 180,E1 -21731.543,E2 -21731.543} C_VEL
LIN {X 0,Y 232.915,Z 510.765,A -85,B 0,C 180,E1 -21732.391,E2 -21732.391} C_VEL
LIN {X 0,Y 234.554,Z 496.882,A -85,B 0,C 180,E1 -21732.972,E2 -21732.972} C_VEL
LIN {X 0,Y 238.348,Z 436.017,A -85,B 0,C 180,E1 -21734.672,E2 -21734.672} C_VEL
LIN {X 0,Y 232.965,Z 423.146,A -85,B 0,C 180,E1 -21736.713,E2 -21736.713} C_VEL
LIN {X 0,Y 226.8,Z 410.643,A -85,B 0,C 180,E1 -21739.179,E2 -21739.179} C_VEL
LIN {X 0,Y 220.479,Z 399.169,A -85,B 0,C 180,E1 -21741.94,E2 -21741.94} C_VEL
LIN {X 0,Y 214.126,Z 388.819,A -85,B 0,C 180,E1 -21745.028,E2 -21745.028} C_VEL
LIN {X 0,Y 210.105,Z 382.839,A -85,B 0,C 180,E1 -21747.199,E2 -21747.199} C_VEL
LIN {X 0,Y 206.768,Z 378.01,A -85,B 0,C 180,E1 -21749.176,E2 -21749.176} C_VEL
LIN {X 0,Y 202.621,Z 372.36,A -85,B 0,C 180,E1 -21751.901,E2 -21751.901} C_VEL
LIN {X 0,Y 201.652,Z 371.318,A -85,B 0,C 180,E1 -21752.572,E2 -21752.572} C_VEL
LIN {X 0,Y 199.147,Z 369.039,A -85,B 0,C 180,E1 -21754.386,E2 -21754.386} C_VEL
LIN {X 0,Y 197.699,Z 366.257,A -85,B 0,C 180,E1 -21755.666,E2 -21755.666} C_VEL
LIN {X 0,Y 194.263,Z 363.865,A -85,B 0,C 180,E1 -21758.652,E2 -21758.652} C_VEL
LIN {X 0,Y 192.919,Z 361.449,A -85,B 0,C 180,E1 -21760.169,E2 -21760.169} C_VEL
LIN {X 0,Y 192.629,Z 360.107,A -85,B 0,C 180,E1 -21760.693,E2 -21760.693} C_VEL
LIN {X 0,Y 192.733,Z 360.095,A -85,B 0,C 180,E1 -21765.212,E2 -21765.212} C_VEL
LIN {X 0,Y 192.94,Z 360.067,A -85,B 0,C 180,E1 -21769.567,E2 -21769.567} C_VEL
LIN {X 0,Y 192.957,Z 360.06,A -85,B 0,C 180,E1 -21773.728,E2 -21773.728} C_VEL
LIN {X 0,Y 193.224,Z 360.025,A -85,B 0,C 180,E1 -21777.916,E2 -21777.916} C_VEL
LIN {X 0,Y 193.406,Z 360.018,A -85,B 0,C 180,E1 -21780.001,E2 -21780.001} C_VEL
LIN {X 0,Y 192.938,Z 360.068,A -85,B 0,C 180,E1 -21784.179,E2 -21784.179} C_VEL
LIN {X 0,Y 193.022,Z 360.054,A -85,B 0,C 180,E1 -21788.375,E2 -21788.375} C_VEL
LIN {X 0,Y 192.785,Z 360.082,A -85,B 0,C 180,E1 -21792.635,E2 -21792.635} C_VEL
LIN {X 0,Y 192.774,Z 360.257,A -85,B 0,C 180,E1 -21793.978,E2 -21793.978} C_VEL
LIN {X 0,Y 193.54,Z 362.638,A -85,B 0,C 180,E1 -21794.995,E2 -21794.995} C_VEL
LIN {X 0,Y 195.584,Z 364.983,A -85,B 0,C 180,E1 -21797.017,E2 -21797.017} C_VEL
LIN {X 0,Y 197.727,Z 366.254,A -85,B 0,C 180,E1 -21798.792,E2 -21798.792} C_VEL
LIN {X 0,Y 199.229,Z 369.169,A -85,B 0,C 180,E1 -21800.118,E2 -21800.118} C_VEL
LIN {X 0,Y 201.485,Z 371.217,A -85,B 0,C 180,E1 -21801.754,E2 -21801.754} C_VEL
LIN {X 0,Y 202.501,Z 372.1,A -85,B 0,C 180,E1 -21802.444,E2 -21802.444} C_VEL
LIN {X 0,Y 204.625,Z 375.29,A -85,B 0,C 180,E1 -21803.914,E2 -21803.914} C_VEL
LIN {X 0,Y 206.766,Z 377.327,A -85,B 0,C 180,E1 -21805.211,E2 -21805.211} C_VEL
LIN {X 0,Y 209.482,Z 381.037,A -85,B 0,C 180,E1 -21806.822,E2 -21806.822} C_VEL
LIN {X 0,Y 210.834,Z 382.658,A -85,B 0,C 180,E1 -21807.565,E2 -21807.565} C_VEL
LIN {X 0,Y 214.637,Z 387.742,A -85,B 0,C 180,E1 -21809.557,E2 -21809.557} C_VEL
LIN {X 0,Y 218.334,Z 392.784,A -85,B 0,C 180,E1 -21811.337,E2 -21811.337} C_VEL
LIN {X 0,Y 225.04,Z 402.601,A -85,B 0,C 180,E1 -21814.272,E2 -21814.272} C_VEL
LIN {X 0,Y 230.501,Z 411.577,A -85,B 0,C 180,E1 -21816.454,E2 -21816.454} C_VEL
LIN {X 0,Y 236.286,Z 423.287,A -85,B 0,C 180,E1 -21818.655,E2 -21818.655} C_VEL
LIN {X 0,Y 238.814,Z 428.806,A -85,B 0,C 180,E1 -21819.572,E2 -21819.572} C_VEL
LIN {X 0,Y 234.808,Z 490.313,A -85,B 0,C 180,E1 -21821.283,E2 -21821.283} C_VEL
LIN {X 0,Y 233.059,Z 504.471,A -85,B 0,C 180,E1 -21821.97,E2 -21821.97} C_VEL
LIN {X 0,Y 230.517,Z 518.553,A -85,B 0,C 180,E1 -21822.972,E2 -21822.972} C_VEL
LIN {X 0,Y 227.615,Z 530.714,A -85,B 0,C 180,E1 -21824.122,E2 -21824.122} C_VEL
LIN {X 0,Y 223.835,Z 543.511,A -85,B 0,C 180,E1 -21825.686,E2 -21825.686} C_VEL
LIN {X 0,Y 219.821,Z 554.94,A -85,B 0,C 180,E1 -21827.468,E2 -21827.468} C_VEL
LIN {X 0,Y 215.853,Z 564.764,A -85,B 0,C 180,E1 -21829.37,E2 -21829.37} C_VEL
LIN {X 0,Y 211.252,Z 575.455,A -85,B 0,C 180,E1 -21832.016,E2 -21832.016} C_VEL
LIN {X 0,Y 207.042,Z 584.245,A -85,B 0,C 180,E1 -21834.757,E2 -21834.757} C_VEL
LIN {X 0,Y 202.784,Z 592.646,A -85,B 0,C 180,E1 -21838.095,E2 -21838.095} C_VEL
LIN {X 0,Y 199.049,Z 599.36,A -85,B 0,C 180,E1 -21841.535,E2 -21841.535} C_VEL
LIN {X 0,Y 195.621,Z 605.279,A -85,B 0,C 180,E1 -21845.597,E2 -21845.597} C_VEL
LIN {X 0,Y 193.665,Z 608.689,A -85,B 0,C 180,E1 -21848.722,E2 -21848.722} C_VEL
LIN {X 0,Y 191.781,Z 611.885,A -85,B 0,C 180,E1 -21852.953,E2 -21852.953} C_VEL
LIN {X 0,Y 190.53,Z 613.677,A -85,B 0,C 180,E1 -21857.214,E2 -21857.214} C_VEL
LIN {X 0,Y 190.123,Z 614.127,A -85,B 0,C 180,E1 -21861.497,E2 -21861.497} C_VEL
LIN {X 0,Y 190.242,Z 613.194,A -85,B 0,C 180,E1 -21865.919,E2 -21865.919} C_VEL
LIN {X 0,Y 190.468,Z 611.067,A -85,B 0,C 180,E1 -21870,E2 -21870} C_VEL
LIN {X 0,Y 191.19,Z 607.508,A -85,B 0,C 180,E1 -21874.216,E2 -21874.216} C_VEL
LIN {X 0,Y 192.635,Z 602.467,A -85,B 0,C 180,E1 -21878.391,E2 -21878.391} C_VEL
LIN {X 0,Y 194.257,Z 597.581,A -85,B 0,C 180,E1 -21881.477,E2 -21881.477} C_VEL
LIN {X 0,Y 196.344,Z 591.678,A -85,B 0,C 180,E1 -21884.51,E2 -21884.51} C_VEL
LIN {X 0,Y 198.816,Z 584.595,A -85,B 0,C 180,E1 -21887.484,E2 -21887.484} C_VEL
LIN {X 0,Y 201.679,Z 576.073,A -85,B 0,C 180,E1 -21890.393,E2 -21890.393} C_VEL
LIN {X 0,Y 205.104,Z 565.741,A -85,B 0,C 180,E1 -21893.206,E2 -21893.206} C_VEL
LIN {X 0,Y 208.556,Z 554.197,A -85,B 0,C 180,E1 -21895.712,E2 -21895.712} C_VEL
LIN {X 0,Y 211.663,Z 542.654,A -85,B 0,C 180,E1 -21897.7,E2 -21897.7} C_VEL
LIN {X 0,Y 214.545,Z 529.98,A -85,B 0,C 180,E1 -21899.429,E2 -21899.429} C_VEL
LIN {X 0,Y 217.16,Z 516.811,A -85,B 0,C 180,E1 -21900.779,E2 -21900.779} C_VEL
LIN {X 0,Y 219.218,Z 502.539,A -85,B 0,C 180,E1 -21901.868,E2 -21901.868} C_VEL
LIN {X 0,Y 220.543,Z 488.257,A -85,B 0,C 180,E1 -21902.597,E2 -21902.597} C_VEL
LIN {X 0,Y 224.301,Z 415.648,A -85,B 0,C 180,E1 -21904.792,E2 -21904.792} C_VEL
LIN {X 0,Y 218.479,Z 401.523,A -85,B 0,C 180,E1 -21906.599,E2 -21906.599} C_VEL
LIN {X 0,Y 210.305,Z 387.043,A -85,B 0,C 180,E1 -21909.152,E2 -21909.152} C_VEL
LIN {X 0,Y 203.891,Z 377.087,A -85,B 0,C 180,E1 -21911.313,E2 -21911.313} C_VEL
LIN {X 0,Y 200.879,Z 372.812,A -85,B 0,C 180,E1 -21912.386,E2 -21912.386} C_VEL
LIN {X 0,Y 198.494,Z 369.382,A -85,B 0,C 180,E1 -21913.276,E2 -21913.276} C_VEL
LIN {X 0,Y 196.174,Z 366.107,A -85,B 0,C 180,E1 -21914.173,E2 -21914.173} C_VEL
LIN {X 0,Y 195.409,Z 365,A -85,B 0,C 180,E1 -21914.479,E2 -21914.479} C_VEL
LIN {X 0,Y 193.365,Z 362.689,A -85,B 0,C 180,E1 -21915.279,E2 -21915.279} C_VEL
LIN {X 0,Y 192.508,Z 360.126,A -85,B 0,C 180,E1 -21915.772,E2 -21915.772} C_VEL
LIN {X 0,Y 192.516,Z 360.13,A -85,B 0,C 180,E1 -21920.05,E2 -21920.05} C_VEL
LIN {X 0,Y 192.559,Z 360.125,A -85,B 0,C 180,E1 -21924.269,E2 -21924.269} C_VEL
LIN {X 0,Y 192.605,Z 360.106,A -85,B 0,C 180,E1 -21927.058,E2 -21927.058} C_VEL
LIN {X 0,Y 192.657,Z 360.09,A -85,B 0,C 180,E1 -21931.69,E2 -21931.69} C_VEL
LIN {X 0,Y 192.67,Z 360.111,A -85,B 0,C 180,E1 -21936.343,E2 -21936.343} C_VEL
LIN {X 0,Y 192.69,Z 360.091,A -85,B 0,C 180,E1 -21941.49,E2 -21941.49} C_VEL
LIN {X 0,Y 192.723,Z 360.089,A -85,B 0,C 180,E1 -21945.21,E2 -21945.21} C_VEL
LIN {X 0,Y 192.941,Z 360.061,A -85,B 0,C 180,E1 -21949.566,E2 -21949.566} C_VEL
LIN {X 0,Y 192.964,Z 360.051,A -85,B 0,C 180,E1 -21953.726,E2 -21953.726} C_VEL
LIN {X 0,Y 193.225,Z 360.028,A -85,B 0,C 180,E1 -21957.915,E2 -21957.915} C_VEL
LIN {X 0,Y 193.402,Z 360.02,A -85,B 0,C 180,E1 -21959.999,E2 -21959.999} C_VEL
LIN {X 0,Y 192.909,Z 360.064,A -85,B 0,C 180,E1 -21964.178,E2 -21964.178} C_VEL
LIN {X 0,Y 193.014,Z 360.052,A -85,B 0,C 180,E1 -21968.374,E2 -21968.374} C_VEL
LIN {X 0,Y 192.783,Z 360.097,A -85,B 0,C 180,E1 -21972.634,E2 -21972.634} C_VEL
LIN {X 0,Y 192.713,Z 360.093,A -85,B 0,C 180,E1 -21976.962,E2 -21976.962} C_VEL
LIN {X 0,Y 192.594,Z 360.101,A -85,B 0,C 180,E1 -21981.402,E2 -21981.402} C_VEL
LIN {X 0,Y 192.634,Z 360.111,A -85,B 0,C 180,E1 -21984.207,E2 -21984.207} C_VEL
LIN {X 0,Y 192.596,Z 360.117,A -85,B 0,C 180,E1 -21988.866,E2 -21988.866} C_VEL
LIN {X 0,Y 192.59,Z 360.116,A -85,B 0,C 180,E1 -21993.187,E2 -21993.187} C_VEL
LIN {X 0,Y 192.541,Z 360.154,A -85,B 0,C 180,E1 -21997.745,E2 -21997.745} C_VEL
LIN {X 0,Y 192.663,Z 360.897,A -85,B 0,C 180,E1 -21998.02,E2 -21998.02} C_VEL
LIN {X 0,Y 193.925,Z 363.506,A -85,B 0,C 180,E1 -21998.59,E2 -21998.59} C_VEL
LIN {X 0,Y 196.458,Z 366.468,A -85,B 0,C 180,E1 -21999.575,E2 -21999.575} C_VEL
LIN {X 0,Y 203.265,Z 377.804,A -85,B 0,C 180,E1 -22002.184,E2 -22002.184} C_VEL
LIN {X 0,Y 209.501,Z 389.006,A -85,B 0,C 180,E1 -22004.371,E2 -22004.371} C_VEL
LIN {X 0,Y 216.141,Z 403.027,A -85,B 0,C 180,E1 -22006.58,E2 -22006.58} C_VEL
LIN {X 0,Y 219.155,Z 410.12,A -85,B 0,C 180,E1 -22007.546,E2 -22007.546} C_VEL
LIN {X 0,Y 219.879,Z 413.794,A -85,B 0,C 180,E1 -22007.853,E2 -22007.853} C_VEL
LIN {X 0,Y 219.87,Z 417.717,A -85,B 0,C 180,E1 -22008.014,E2 -22008.014} C_VEL
LIN {X 0,Y 218.131,Z 431.246,A -85,B 0,C 180,E1 -22008.205,E2 -22008.205} C_VEL
LIN {X 0,Y 214.235,Z 499.893,A -85,B 0,C 180,E1 -22010.308,E2 -22010.308} C_VEL
LIN {X 0,Y 212.658,Z 513.651,A -85,B 0,C 180,E1 -22011.029,E2 -22011.029} C_VEL
LIN {X 0,Y 210.355,Z 527.786,A -85,B 0,C 180,E1 -22012.128,E2 -22012.128} C_VEL
LIN {X 0,Y 207.344,Z 541.768,A -85,B 0,C 180,E1 -22013.619,E2 -22013.619} C_VEL
LIN {X 0,Y 204.185,Z 554.289,A -85,B 0,C 180,E1 -22015.395,E2 -22015.395} C_VEL
LIN {X 0,Y 200.74,Z 566.223,A -85,B 0,C 180,E1 -22017.558,E2 -22017.558} C_VEL
LIN {X 0,Y 197.117,Z 577.205,A -85,B 0,C 180,E1 -22020.057,E2 -22020.057} C_VEL
LIN {X 0,Y 193.523,Z 587.434,A -85,B 0,C 180,E1 -22023.003,E2 -22023.003} C_VEL
LIN {X 0,Y 190.519,Z 595.921,A -85,B 0,C 180,E1 -22026.061,E2 -22026.061} C_VEL
LIN {X 0,Y 187.798,Z 603.615,A -85,B 0,C 180,E1 -22029.521,E2 -22029.521} C_VEL
LIN {X 0,Y 186.173,Z 608.843,A -85,B 0,C 180,E1 -22032.423,E2 -22032.423} C_VEL
LIN {X 0,Y 184.68,Z 613.639,A -85,B 0,C 180,E1 -22035.679,E2 -22035.679} C_VEL
LIN {X 0,Y 183.533,Z 618.599,A -85,B 0,C 180,E1 -22040.078,E2 -22040.078} C_VEL
LIN {X 0,Y 183.134,Z 621.307,A -85,B 0,C 180,E1 -22043.389,E2 -22043.389} C_VEL
LIN {X 0,Y 183.051,Z 623.169,A -85,B 0,C 180,E1 -22046.586,E2 -22046.586} C_VEL
LIN {X 0,Y 183.185,Z 624.329,A -85,B 0,C 180,E1 -22050,E2 -22050} C_VEL
LIN {X 0,Y 183.031,Z 624.63,A -85,B 0,C 180,E1 -22054.404,E2 -22054.404} C_VEL
LIN {X 0,Y 183.4,Z 623.604,A -85,B 0,C 180,E1 -22058.817,E2 -22058.817} C_VEL
LIN {X 0,Y 184.464,Z 621.245,A -85,B 0,C 180,E1 -22063.214,E2 -22063.214} C_VEL
LIN {X 0,Y 186.542,Z 617.499,A -85,B 0,C 180,E1 -22067.541,E2 -22067.541} C_VEL
LIN {X 0,Y 189.399,Z 612.259,A -85,B 0,C 180,E1 -22071.781,E2 -22071.781} C_VEL
LIN {X 0,Y 192.264,Z 607.2,A -85,B 0,C 180,E1 -22074.857,E2 -22074.857} C_VEL
LIN {X 0,Y 196.29,Z 599.999,A -85,B 0,C 180,E1 -22078.32,E2 -22078.32} C_VEL
LIN {X 0,Y 201.044,Z 591.122,A -85,B 0,C 180,E1 -22081.624,E2 -22081.624} C_VEL
LIN {X 0,Y 205.72,Z 581.832,A -85,B 0,C 180,E1 -22084.31,E2 -22084.31} C_VEL
LIN {X 0,Y 209.904,Z 572.358,A -85,B 0,C 180,E1 -22086.529,E2 -22086.529} C_VEL
LIN {X 0,Y 214.293,Z 561.535,A -85,B 0,C 180,E1 -22088.544,E2 -22088.544} C_VEL
LIN {X 0,Y 218.58,Z 549.404,A -85,B 0,C 180,E1 -22090.32,E2 -22090.32} C_VEL
LIN {X 0,Y 222.087,Z 537.754,A -85,B 0,C 180,E1 -22091.646,E2 -22091.646} C_VEL
LIN {X 0,Y 225.504,Z 523.903,A -85,B 0,C 180,E1 -22092.827,E2 -22092.827} C_VEL
LIN {X 0,Y 228.031,Z 510.129,A -85,B 0,C 180,E1 -22093.674,E2 -22093.674} C_VEL
LIN {X 0,Y 229.699,Z 495.978,A -85,B 0,C 180,E1 -22094.264,E2 -22094.264} C_VEL
LIN {X 0,Y 233.432,Z 438.333,A -85,B 0,C 180,E1 -22095.886,E2 -22095.886} C_VEL
LIN {X 0,Y 228.369,Z 426.258,A -85,B 0,C 180,E1 -22097.92,E2 -22097.92} C_VEL
LIN {X 0,Y 222.919,Z 415.026,A -85,B 0,C 180,E1 -22100.232,E2 -22100.232} C_VEL
LIN {X 0,Y 217.099,Z 404.209,A -85,B 0,C 180,E1 -22102.92,E2 -22102.92} C_VEL
LIN {X 0,Y 211.451,Z 394.714,A -85,B 0,C 180,E1 -22105.813,E2 -22105.813} C_VEL
LIN {X 0,Y 207.545,Z 388.743,A -85,B 0,C 180,E1 -22108.026,E2 -22108.026} C_VEL
LIN {X 0,Y 204.281,Z 383.915,A -85,B 0,C 180,E1 -22110.059,E2 -22110.059} C_VEL
LIN {X 0,Y 200.091,Z 378.099,A -85,B 0,C 180,E1 -22112.973,E2 -22112.973} C_VEL
LIN {X 0,Y 197.379,Z 375.582,A -85,B 0,C 180,E1 -22115.007,E2 -22115.007} C_VEL
LIN {X 0,Y 195.823,Z 372.751,A -85,B 0,C 180,E1 -22116.428,E2 -22116.428} C_VEL
LIN {X 0,Y 192.798,Z 370.577,A -85,B 0,C 180,E1 -22119.182,E2 -22119.182} C_VEL
LIN {X 0,Y 191.197,Z 367.643,A -85,B 0,C 180,E1 -22121.093,E2 -22121.093} C_VEL
LIN {X 0,Y 191.043,Z 367.114,A -85,B 0,C 180,E1 -22121.323,E2 -22121.323} C_VEL
LIN {X 0,Y 187.615,Z 365.026,A -85,B 0,C 180,E1 -22125.908,E2 -22125.908} C_VEL
LIN {X 0,Y 186.204,Z 362.473,A -85,B 0,C 180,E1 -22128.974,E2 -22128.974} C_VEL
LIN {X 0,Y 185.905,Z 360.95,A -85,B 0,C 180,E1 -22130.249,E2 -22130.249} C_VEL
LIN {X 0,Y 185.922,Z 360.935,A -85,B 0,C 180,E1 -22133.489,E2 -22133.489} C_VEL
LIN {X 0,Y 186.17,Z 360.903,A -85,B 0,C 180,E1 -22137.837,E2 -22137.837} C_VEL
LIN {X 0,Y 186.372,Z 360.894,A -85,B 0,C 180,E1 -22140.001,E2 -22140.001} C_VEL
LIN {X 0,Y 185.907,Z 361.1,A -85,B 0,C 180,E1 -22144.405,E2 -22144.405} C_VEL
LIN {X 0,Y 186.738,Z 363.488,A -85,B 0,C 180,E1 -22146.755,E2 -22146.755} C_VEL
LIN {X 0,Y 189.463,Z 366.315,A -85,B 0,C 180,E1 -22151.231,E2 -22151.231} C_VEL
LIN {X 0,Y 191.194,Z 367.195,A -85,B 0,C 180,E1 -22153.283,E2 -22153.283} C_VEL
LIN {X 0,Y 192.409,Z 369.89,A -85,B 0,C 180,E1 -22154.815,E2 -22154.815} C_VEL
LIN {X 0,Y 194.736,Z 372.181,A -85,B 0,C 180,E1 -22157.094,E2 -22157.094} C_VEL
LIN {X 0,Y 195.965,Z 373.018,A -85,B 0,C 180,E1 -22158.144,E2 -22158.144} C_VEL
LIN {X 0,Y 197.822,Z 376.157,A -85,B 0,C 180,E1 -22159.793,E2 -22159.793} C_VEL
LIN {X 0,Y 200.482,Z 378.584,A -85,B 0,C 180,E1 -22161.75,E2 -22161.75} C_VEL
LIN {X 0,Y 202.983,Z 382.096,A -85,B 0,C 180,E1 -22163.519,E2 -22163.519} C_VEL
LIN {X 0,Y 204.61,Z 383.767,A -85,B 0,C 180,E1 -22164.545,E2 -22164.545} C_VEL
LIN {X 0,Y 207.563,Z 387.655,A -85,B 0,C 180,E1 -22166.345,E2 -22166.345} C_VEL
LIN {X 0,Y 212.217,Z 394.034,A -85,B 0,C 180,E1 -22168.916,E2 -22168.916} C_VEL
LIN {X 0,Y 217.219,Z 401.031,A -85,B 0,C 180,E1 -22171.38,E2 -22171.38} C_VEL
LIN {X 0,Y 224.219,Z 411.998,A -85,B 0,C 180,E1 -22174.484,E2 -22174.484} C_VEL
LIN {X 0,Y 227.788,Z 418.418,A -85,B 0,C 180,E1 -22175.956,E2 -22175.956} C_VEL
LIN {X 0,Y 233.311,Z 430.021,A -85,B 0,C 180,E1 -22178.138,E2 -22178.138} C_VEL
LIN {X 0,Y 233.883,Z 431.337,A -85,B 0,C 180,E1 -22178.358,E2 -22178.358} C_VEL
LIN {X 0,Y 229.909,Z 490.334,A -85,B 0,C 180,E1 -22180.016,E2 -22180.016} C_VEL
LIN {X 0,Y 228.063,Z 504.801,A -85,B 0,C 180,E1 -22180.724,E2 -22180.724} C_VEL
LIN {X 0,Y 225.421,Z 518.848,A -85,B 0,C 180,E1 -22181.731,E2 -22181.731} C_VEL
LIN {X 0,Y 222.193,Z 531.884,A -85,B 0,C 180,E1 -22182.994,E2 -22182.994} C_VEL
LIN {X 0,Y 218.278,Z 544.493,A -85,B 0,C 180,E1 -22184.574,E2 -22184.574} C_VEL
LIN {X 0,Y 214.056,Z 555.967,A -85,B 0,C 180,E1 -22186.412,E2 -22186.412} C_VEL
LIN {X 0,Y 209.568,Z 566.481,A -85,B 0,C 180,E1 -22188.524,E2 -22188.524} C_VEL
LIN {X 0,Y 204.831,Z 576.914,A -85,B 0,C 180,E1 -22191.233,E2 -22191.233} C_VEL
LIN {X 0,Y 200.499,Z 585.489,A -85,B 0,C 180,E1 -22194.048,E2 -22194.048} C_VEL
LIN {X 0,Y 196.078,Z 593.644,A -85,B 0,C 180,E1 -22197.478,E2 -22197.478} C_VEL
LIN {X 0,Y 192.715,Z 599.364,A -85,B 0,C 180,E1 -22200.507,E2 -22200.507} C_VEL
LIN {X 0,Y 189.071,Z 605.338,A -85,B 0,C 180,E1 -22204.694,E2 -22204.694} C_VEL
LIN {X 0,Y 186.937,Z 608.77,A -85,B 0,C 180,E1 -22207.917,E2 -22207.917} C_VEL
LIN {X 0,Y 184.9,Z 612.021,A -85,B 0,C 180,E1 -22212.298,E2 -22212.298} C_VEL
LIN {X 0,Y 183.534,Z 613.852,A -85,B 0,C 180,E1 -22216.718,E2 -22216.718} C_VEL
LIN {X 0,Y 183.028,Z 614.34,A -85,B 0,C 180,E1 -22221.165,E2 -22221.165} C_VEL
LIN {X 0,Y 183.123,Z 613.503,A -85,B 0,C 180,E1 -22225.598,E2 -22225.598} C_VEL
LIN {X 0,Y 183.381,Z 611.352,A -85,B 0,C 180,E1 -22230,E2 -22230} C_VEL
LIN {X 0,Y 184.124,Z 607.833,A -85,B 0,C 180,E1 -22234.378,E2 -22234.378} C_VEL
LIN {X 0,Y 185.631,Z 602.833,A -85,B 0,C 180,E1 -22238.71,E2 -22238.71} C_VEL
LIN {X 0,Y 187.329,Z 597.991,A -85,B 0,C 180,E1 -22241.908,E2 -22241.908} C_VEL
LIN {X 0,Y 189.511,Z 592.136,A -85,B 0,C 180,E1 -22245.046,E2 -22245.046} C_VEL
LIN {X 0,Y 192.472,Z 583.9,A -85,B 0,C 180,E1 -22248.577,E2 -22248.577} C_VEL
LIN {X 0,Y 195.63,Z 575.034,A -85,B 0,C 180,E1 -22251.606,E2 -22251.606} C_VEL
LIN {X 0,Y 199.258,Z 564.454,A -85,B 0,C 180,E1 -22254.483,E2 -22254.483} C_VEL
LIN {X 0,Y 202.591,Z 553.768,A -85,B 0,C 180,E1 -22256.806,E2 -22256.806} C_VEL
LIN {X 0,Y 205.838,Z 542.088,A -85,B 0,C 180,E1 -22258.833,E2 -22258.833} C_VEL
LIN {X 0,Y 208.425,Z 530.987,A -85,B 0,C 180,E1 -22260.383,E2 -22260.383} C_VEL
LIN {X 0,Y 211.106,Z 518.047,A -85,B 0,C 180,E1 -22261.763,E2 -22261.763} C_VEL
LIN {X 0,Y 213.278,Z 504.136,A -85,B 0,C 180,E1 -22262.865,E2 -22262.865} C_VEL
LIN {X 0,Y 214.753,Z 489.594,A -85,B 0,C 180,E1 -22263.661,E2 -22263.661} C_VEL
LIN {X 0,Y 218.696,Z 417.738,A -85,B 0,C 180,E1 -22265.872,E2 -22265.872} C_VEL
LIN {X 0,Y 213.603,Z 405.304,A -85,B 0,C 180,E1 -22267.542,E2 -22267.542} C_VEL
LIN {X 0,Y 204.944,Z 389.83,A -85,B 0,C 180,E1 -22270.412,E2 -22270.412} C_VEL
LIN {X 0,Y 197.507,Z 378.549,A -85,B 0,C 180,E1 -22273.103,E2 -22273.103} C_VEL
LIN {X 0,Y 194.421,Z 374.243,A -85,B 0,C 180,E1 -22274.302,E2 -22274.302} C_VEL
LIN {X 0,Y 191.797,Z 370.489,A -85,B 0,C 180,E1 -22275.378,E2 -22275.378} C_VEL
LIN {X 0,Y 189.468,Z 367.384,A -85,B 0,C 180,E1 -22276.366,E2 -22276.366} C_VEL
LIN {X 0,Y 188.63,Z 366.092,A -85,B 0,C 180,E1 -22276.743,E2 -22276.743} C_VEL
LIN {X 0,Y 186.479,Z 363.938,A -85,B 0,C 180,E1 -22277.669,E2 -22277.669} C_VEL
LIN {X 0,Y 185.532,Z 361.552,A -85,B 0,C 180,E1 -22278.177,E2 -22278.177} C_VEL
LIN {X 0,Y 185.434,Z 361.003,A -85,B 0,C 180,E1 -22278.304,E2 -22278.304} C_VEL
LIN {X 0,Y 185.504,Z 360.993,A -85,B 0,C 180,E1 -22282.71,E2 -22282.71} C_VEL
LIN {X 0,Y 185.54,Z 360.991,A -85,B 0,C 180,E1 -22287.973,E2 -22287.973} C_VEL
LIN {X 0,Y 185.578,Z 360.982,A -85,B 0,C 180,E1 -22290.575,E2 -22290.575} C_VEL
LIN {X 0,Y 185.577,Z 360.992,A -85,B 0,C 180,E1 -22295.38,E2 -22295.38} C_VEL
LIN {X 0,Y 185.621,Z 360.967,A -85,B 0,C 180,E1 -22301.178,E2 -22301.178} C_VEL
LIN {X 0,Y 185.655,Z 360.976,A -85,B 0,C 180,E1 -22304.633,E2 -22304.633} C_VEL
LIN {X 0,Y 185.884,Z 360.938,A -85,B 0,C 180,E1 -22309.418,E2 -22309.418} C_VEL
LIN {X 0,Y 185.929,Z 360.93,A -85,B 0,C 180,E1 -22313.488,E2 -22313.488} C_VEL
LIN {X 0,Y 186.172,Z 360.904,A -85,B 0,C 180,E1 -22317.836,E2 -22317.836} C_VEL
LIN {X 0,Y 186.367,Z 360.896,A -85,B 0,C 180,E1 -22319.999,E2 -22319.999} C_VEL
LIN {X 0,Y 185.918,Z 360.952,A -85,B 0,C 180,E1 -22326.511,E2 -22326.511} C_VEL
LIN {X 0,Y 185.883,Z 360.939,A -85,B 0,C 180,E1 -22330.58,E2 -22330.58} C_VEL
LIN {X 0,Y 185.662,Z 360.965,A -85,B 0,C 180,E1 -22335.365,E2 -22335.365} C_VEL
LIN {X 0,Y 185.537,Z 360.986,A -85,B 0,C 180,E1 -22339.932,E2 -22339.932} C_VEL
LIN {X 0,Y 185.572,Z 360.986,A -85,B 0,C 180,E1 -22344.646,E2 -22344.646} C_VEL
LIN {X 0,Y 185.539,Z 360.99,A -85,B 0,C 180,E1 -22349.499,E2 -22349.499} C_VEL
LIN {X 0,Y 185.494,Z 360.997,A -85,B 0,C 180,E1 -22354.633,E2 -22354.633} C_VEL
LIN {X 0,Y 185.508,Z 361,A -85,B 0,C 180,E1 -22355.375,E2 -22355.375} C_VEL
LIN {X 0,Y 186.53,Z 363.867,A -85,B 0,C 180,E1 -22355.981,E2 -22355.981} C_VEL
LIN {X 0,Y 188.695,Z 366.071,A -85,B 0,C 180,E1 -22356.915,E2 -22356.915} C_VEL
LIN {X 0,Y 191.3,Z 369.998,A -85,B 0,C 180,E1 -22358.061,E2 -22358.061} C_VEL
LIN {X 0,Y 193.165,Z 372.408,A -85,B 0,C 180,E1 -22358.825,E2 -22358.825} C_VEL
LIN {X 0,Y 199.059,Z 382.374,A -85,B 0,C 180,E1 -22361.199,E2 -22361.199} C_VEL
LIN {X 0,Y 205.499,Z 394.299,A -85,B 0,C 180,E1 -22363.584,E2 -22363.584} C_VEL
LIN {X 0,Y 211.361,Z 406.911,A -85,B 0,C 180,E1 -22365.636,E2 -22365.636} C_VEL
LIN {X 0,Y 217.072,Z 421.321,A -85,B 0,C 180,E1 -22367.563,E2 -22367.563} C_VEL
LIN {X 0,Y 218.106,Z 424.621,A -85,B 0,C 180,E1 -22367.925,E2 -22367.925} C_VEL
LIN {X 0,Y 218.246,Z 429.113,A -85,B 0,C 180,E1 -22368.141,E2 -22368.141} C_VEL
LIN {X 0,Y 218.131,Z 431.246,A -85,B 0,C 180,E1 -22368.205,E2 -22368.205} C_VEL
LIN {X 0,Y 217.294,Z 437.088,A -85,B 0,C 180,E1 -22368.271,E2 -22368.271} C_VEL
LIN {X 0,Y 211.714,Z 456.07,A -85,B 0,C 180,E1 -22367.865,E2 -22367.865} C_VEL
LIN {X 0,Y 210.836,Z 461.914,A -85,B 0,C 180,E1 -22367.922,E2 -22367.922} C_VEL
LIN {X 0,Y 208.651,Z 499.136,A -85,B 0,C 180,E1 -22369.108,E2 -22369.108} C_VEL
LIN {X 0,Y 207.045,Z 513.047,A -85,B 0,C 180,E1 -22369.84,E2 -22369.84} C_VEL
LIN {X 0,Y 204.784,Z 526.721,A -85,B 0,C 180,E1 -22370.906,E2 -22370.906} C_VEL
LIN {X 0,Y 202.076,Z 539.11,A -85,B 0,C 180,E1 -22372.196,E2 -22372.196} C_VEL
LIN {X 0,Y 198.697,Z 552.094,A -85,B 0,C 180,E1 -22373.984,E2 -22373.984} C_VEL
LIN {X 0,Y 195.278,Z 563.872,A -85,B 0,C 180,E1 -22376.09,E2 -22376.09} C_VEL
LIN {X 0,Y 192.369,Z 572.702,A -85,B 0,C 180,E1 -22378.013,E2 -22378.013} C_VEL
LIN {X 0,Y 188.306,Z 583.691,A -85,B 0,C 180,E1 -22380.976,E2 -22380.976} C_VEL
LIN {X 0,Y 184.958,Z 592.775,A -85,B 0,C 180,E1 -22384.09,E2 -22384.09} C_VEL
LIN {X 0,Y 182.188,Z 600.334,A -85,B 0,C 180,E1 -22387.31,E2 -22387.31} C_VEL
LIN {X 0,Y 179.997,Z 606.636,A -85,B 0,C 180,E1 -22390.617,E2 -22390.617} C_VEL
LIN {X 0,Y 178.25,Z 611.823,A -85,B 0,C 180,E1 -22393.979,E2 -22393.979} C_VEL
LIN {X 0,Y 177.004,Z 615.996,A -85,B 0,C 180,E1 -22397.387,E2 -22397.387} C_VEL
LIN {X 0,Y 176.324,Z 619.313,A -85,B 0,C 180,E1 -22400.826,E2 -22400.826} C_VEL
LIN {X 0,Y 175.97,Z 622.406,A -85,B 0,C 180,E1 -22405.419,E2 -22405.419} C_VEL
LIN {X 0,Y 176.091,Z 624.105,A -85,B 0,C 180,E1 -22410,E2 -22410} C_VEL
LIN {X 0,Y 175.943,Z 624.435,A -85,B 0,C 180,E1 -22414.582,E2 -22414.582} C_VEL
